   cmSepaGripperAxisZ.commandConfiguration.haltSuperimposed.jerk := -1.0;
   cmSepaGripperAxisZ.commandConfiguration.haltSuperimposed.abortAcceleration := FALSE;
   cmSepaGripperAxisZ.commandConfiguration.gearInRelative.ratioNumerator := 1;
   cmSepaGripperAxisZ.commandConfiguration.gearInRelative.ratioDenominator := 1;
   cmSepaGripperAxisZ.commandConfiguration.gearInRelative.acceleration := -1.0;
   cmSepaGripperAxisZ.commandConfiguration.gearInRelative.deceleration := -1.0;
   cmSepaGripperAxisZ.commandConfiguration.gearInRelative.jerk := -1.0;
   cmSepaGripperAxisZ.commandConfiguration.gearInRelative.ratioChangeOnTheFly := FALSE;
   cmSepaGripperAxisZ.commandConfiguration.gearInAbsolute.ratioNumerator := 1;
   cmSepaGripperAxisZ.commandConfiguration.gearInAbsolute.ratioDenominator := 1;
   cmSepaGripperAxisZ.commandConfiguration.gearInAbsolute.masterSyncPosition := 0.0;
   cmSepaGripperAxisZ.commandConfiguration.gearInAbsolute.slaveSyncPosition := 0.0;
   cmSepaGripperAxisZ.commandConfiguration.gearInAbsolute.syncProfileReference := 1;
   cmSepaGripperAxisZ.commandConfiguration.gearInAbsolute.masterStartDistance := 0.0;
   cmSepaGripperAxisZ.commandConfiguration.gearInAbsolute.velocity := -1.0;
   cmSepaGripperAxisZ.commandConfiguration.gearInAbsolute.acceleration := -1.0;
   cmSepaGripperAxisZ.commandConfiguration.gearInAbsolute.deceleration := -1.0;
   cmSepaGripperAxisZ.commandConfiguration.gearInAbsolute.jerk := -1.0;
   cmSepaGripperAxisZ.commandConfiguration.gearInAbsolute.syncDirection := 1;
   cmSepaGripperAxisZ.commandConfiguration.gearInAbsolute.ratioChangeOnTheFly := FALSE;
   cmSepaGripperAxisZ.commandConfiguration.gearInVelocity.continuousUpdate := FALSE;
   cmSepaGripperAxisZ.commandConfiguration.gearInVelocity.ratioNumerator := 1;
   cmSepaGripperAxisZ.commandConfiguration.gearInVelocity.ratioDenominator := 1;
   cmSepaGripperAxisZ.commandConfiguration.gearInVelocity.acceleration := -1.0;
   cmSepaGripperAxisZ.commandConfiguration.gearInVelocity.deceleration := -1.0;
   cmSepaGripperAxisZ.commandConfiguration.gearInVelocity.jerk := -1.0;
   cmSepaGripperAxisZ.commandConfiguration.gearInVelocity.positionControlled := FALSE;
   cmSepaGripperAxisZ.commandConfiguration.camIn.masterOffset := 0.0;
   cmSepaGripperAxisZ.commandConfiguration.camIn.slaveOffset := 0.0;
   cmSepaGripperAxisZ.commandConfiguration.camIn.masterScaling := 1.0;
   cmSepaGripperAxisZ.commandConfiguration.camIn.slaveScaling := 1.0;
   cmSepaGripperAxisZ.commandConfiguration.camIn.masterSyncPosition := 0.0;
   cmSepaGripperAxisZ.commandConfiguration.camIn.syncProfileReference := 1;
   cmSepaGripperAxisZ.commandConfiguration.camIn.masterStartDistance := 0.0;
   cmSepaGripperAxisZ.commandConfiguration.camIn.velocity := -1.0;
   cmSepaGripperAxisZ.commandConfiguration.camIn.acceleration := -1.0;
   cmSepaGripperAxisZ.commandConfiguration.camIn.deceleration := -1.0;
   cmSepaGripperAxisZ.commandConfiguration.camIn.jerk := -1.0;
   cmSepaGripperAxisZ.commandConfiguration.camIn.applicationMode := 0;
   cmSepaGripperAxisZ.commandConfiguration.camIn.syncDirection := 1;
   cmSepaGripperAxisZ.commandConfiguration.gearOutCamOut.slavePosition := 0.0;
   cmSepaGripperAxisZ.commandConfiguration.gearOutCamOut.syncProfileReference := 1;
   cmSepaGripperAxisZ.commandConfiguration.gearOutCamOut.masterStopDistance := 0.0;
   cmSepaGripperAxisZ.commandConfiguration.gearOutCamOut.deceleration := -1.0;
   cmSepaGripperAxisZ.commandConfiguration.gearOutCamOut.jerk := -1.0;
   cmSepaGripperAxisZ.commandConfiguration.gearOutCamOut.syncOutDirection := 3;
   cmSepaGripperAxisZ.commandConfiguration.gearOutCamOut.gearOutCamOutMode := -1;
   cmSepaGripperAxisZ.commandConfiguration.phasing.phaseShift := 0.0;
   cmSepaGripperAxisZ.commandConfiguration.phasing.velocity := -1.0;
   cmSepaGripperAxisZ.commandConfiguration.phasing.acceleration := -1.0;
   cmSepaGripperAxisZ.commandConfiguration.phasing.deceleration := -1.0;
   cmSepaGripperAxisZ.commandConfiguration.phasing.jerk := -1.0;
   cmSepaGripperAxisZ.commandConfiguration.phasing.profileReference := 0;
   cmSepaGripperAxisZ.commandConfiguration.phasing.phasingDistance := 0.0;
   cmSepaGripperAxisZ.commandConfiguration.phasing.startPosition := 0.0;
   cmSepaGripperAxisZ.commandConfiguration.phasing.direction := 3;
   cmSepaGripperAxisZ.commandConfiguration.phasing.phaseAbsolute := TRUE;
   cmSepaGripperAxisZ.commandConfiguration.phasing.phaseShiftChangeOnTheFly := FALSE;
   cmSepaGripperAxisZ.commandConfiguration.offset.offset := 0.0;
   cmSepaGripperAxisZ.commandConfiguration.offset.profileReference := 1;
   cmSepaGripperAxisZ.commandConfiguration.offset.offsetDistance := 0.0;
   cmSepaGripperAxisZ.commandConfiguration.offset.startPosition := 0.0;
   cmSepaGripperAxisZ.commandConfiguration.offset.direction := 3;
   cmSepaGripperAxisZ.commandConfiguration.offset.offsetAbsolute := TRUE;
   cmSepaGripperAxisZ.commandConfiguration.offset.offsetChangeOnTheFly := FALSE;
   cmSepaGripperAxisZ.commands.enableMasterControl := TRUE;
   cmSepaGripperAxisZ.commands.enableAxis := FALSE;
   cmSepaGripperAxisZ.commands.resetAxis := FALSE;
   cmSepaGripperAxisZ.commands.openBrake := FALSE;
   cmSepaGripperAxisZ.commands.jogForward := FALSE;
   cmSepaGripperAxisZ.commands.jogBackward := FALSE;
   cmSepaGripperAxisZ.commands.moveVelocity := FALSE;
   cmSepaGripperAxisZ.commands.stop := FALSE;
   cmSepaGripperAxisZ.commands.fastStop := FALSE;
   cmSepaGripperAxisZ.commands.torqueLimiting := FALSE;
   cmSepaGripperAxisZ.commands.homing := FALSE;
   cmSepaGripperAxisZ.commands.posRelative := FALSE;
   cmSepaGripperAxisZ.commands.posAbsolute := FALSE;
   cmSepaGripperAxisZ.commands.posSuperimposed := FALSE;
   cmSepaGripperAxisZ.commands.haltSuperimposed := FALSE;
   cmSepaGripperAxisZ.commands.selectSetPosition := -1;
   cmSepaGripperAxisZ.commands.uploadParameters := FALSE;
   cmSepaGripperAxisZ.commands.refreshConfiguration := FALSE;
   cmSepaGripperAxisZ.commands.editConfiguration := FALSE;
   cmSepaGripperAxisZ.commands.saveConfiguration := FALSE;
   cmSepaGripperAxisZ.commands.uploadCurrentTorque := FALSE;
   cmSepaGripperAxisZ.commands.reset := FALSE;
   cmSepaGripperAxisZ.monitoring.enable := TRUE;
   cmSepaGripperAxisZ.monitoring.referenceDesignator := WSTRING#'SepaGripperAxisZ';
   cmSepaGripperAxisZ.monitoring.enabled := TRUE;
   cmSepaGripperAxisZ.monitoring.enableManualCmds := FALSE;
   cmSepaGripperAxisZ.monitoring.reset := FALSE;
   cmSepaGripperAxisZ.monitoring.resetAxis := FALSE;
   cmSepaGripperAxisZ.monitoring.enableAxis := TRUE;
   cmSepaGripperAxisZ.monitoring.openBrake := FALSE;
   cmSepaGripperAxisZ.monitoring.jogBackward := FALSE;
   cmSepaGripperAxisZ.monitoring.jogForward := FALSE;
   cmSepaGripperAxisZ.monitoring.moveVelocity := FALSE;
   cmSepaGripperAxisZ.monitoring.stop := FALSE;
   cmSepaGripperAxisZ.monitoring.fastStop := FALSE;
   cmSepaGripperAxisZ.monitoring.torqueLimiting := FALSE;
   cmSepaGripperAxisZ.monitoring.homing := FALSE;
   cmSepaGripperAxisZ.monitoring.posRelative := FALSE;
   cmSepaGripperAxisZ.monitoring.posAbsolute := FALSE;
   cmSepaGripperAxisZ.monitoring.posSuperimposed := FALSE;
   cmSepaGripperAxisZ.monitoring.haltSuperimposed := FALSE;
   cmSepaGripperAxisZ.monitoring.brakeOpened := FALSE;
   cmSepaGripperAxisZ.monitoring.axisEnabled := TRUE;
   cmSepaGripperAxisZ.monitoring.resetActive := FALSE;
   cmSepaGripperAxisZ.monitoring.inVelocity := FALSE;
   cmSepaGripperAxisZ.monitoring.inLimitation := FALSE;
   cmSepaGripperAxisZ.monitoring.inClamping := FALSE;
   cmSepaGripperAxisZ.monitoring.startSync := FALSE;
   cmSepaGripperAxisZ.monitoring.inSync := FALSE;
   cmSepaGripperAxisZ.monitoring.inSimulation := FALSE;
   cmSepaGripperAxisZ.monitoring.jogSelected := FALSE;
   cmSepaGripperAxisZ.monitoring.moveVelocitySelected := FALSE;
   cmSepaGripperAxisZ.monitoring.stopSelected := FALSE;
   cmSepaGripperAxisZ.monitoring.fastStopSelected := FALSE;
   cmSepaGripperAxisZ.monitoring.torqueLimitingSelected := FALSE;
   cmSepaGripperAxisZ.monitoring.homingSelected := FALSE;
   cmSepaGripperAxisZ.monitoring.posRelativeSelected := FALSE;
   cmSepaGripperAxisZ.monitoring.posAbsoluteSelected := FALSE;
   cmSepaGripperAxisZ.monitoring.posSuperimposedSelected := FALSE;
   cmSepaGripperAxisZ.monitoring.haltSuperimposedSelected := FALSE;
   cmSepaGripperAxisZ.monitoring.commandBusy := FALSE;
   cmSepaGripperAxisZ.monitoring.commandDone := FALSE;
   cmSepaGripperAxisZ.monitoring.commandAborted := FALSE;
   cmSepaGripperAxisZ.monitoring.homingCommandBusy := FALSE;
   cmSepaGripperAxisZ.monitoring.homingCommandDone := FALSE;
   cmSepaGripperAxisZ.monitoring.homingCommandAborted := FALSE;
   cmSepaGripperAxisZ.monitoring.superimposedBusy := FALSE;
   cmSepaGripperAxisZ.monitoring.superimposedDone := FALSE;
   cmSepaGripperAxisZ.monitoring.superimposedAborted := FALSE;
   cmSepaGripperAxisZ.monitoring.selectSetPosition := -1;
   cmSepaGripperAxisZ.monitoring.selectionController := FALSE;
   cmSepaGripperAxisZ.monitoring.interlockGeneral := TRUE;
   cmSepaGripperAxisZ.monitoring.interlockJogForward := TRUE;
   cmSepaGripperAxisZ.monitoring.interlockJogBackward := TRUE;
   cmSepaGripperAxisZ.monitoring.interlockWarningGeneral := FALSE;
   cmSepaGripperAxisZ.monitoring.interlockWarningJogForward := FALSE;
   cmSepaGripperAxisZ.monitoring.interlockWarningJogBackward := FALSE;
   cmSepaGripperAxisZ.monitoring.valid := TRUE;
   cmSepaGripperAxisZ.monitoring.busy := TRUE;
   cmSepaGripperAxisZ.monitoring.error := FALSE;
   cmSepaGripperAxisZ.monitoring.status := 16#7002;
   cmSepaGripperAxisZ.monitoring.subfunctionStatus := 16#0000;
   cmSepaGripperAxisZ.monitoring.actualPosition := 0.0;
   cmSepaGripperAxisZ.monitoring.actualSpeed := 0.0;
   cmSepaGripperAxisZ.monitoring.speedUnit := 1062;
   cmSepaGripperAxisZ.monitoring.positionUnit := 1013;
   cmSepaGripperAxisZ.monitoring.axisStatus1 := 16#0200_10E1;
   cmSepaGripperAxisZ.monitoring.axisStatus2 := 16#0000_0000;
   cmSepaGripperAxisZ.monitoring.axisType := 1;
   cmSepaGripperAxisZ.monitoring.maxVelocity := 2500.0;
   cmSepaGripperAxisZ.monitoring.actualCurrent := 0.0;
   cmSepaGripperAxisZ.monitoring.actualTorque := 0.0;
   cmSepaGripperAxisZ.monitoring.velocityOverrideEnabled := FALSE;
   cmSepaGripperAxisZ.monitoring.sinaParaError := FALSE;
   cmSepaGripperAxisZ.monitoring.sinaParaStatus := 16#0000_0000;
   cmSepaGripperAxisZ.configuration.referenceDesignator := WSTRING#'SepaGripperAxisZ';
   cmSepaGripperAxisZ.configuration.disableAlarms := FALSE;
   cmSepaGripperAxisZ.configuration.masterControlPopUp := TRUE;
   cmSepaGripperAxisZ.configuration.setPositions[0].position := 0.0;
   cmSepaGripperAxisZ.configuration.setPositions[1].position := 25.0;
   cmSepaGripperAxisZ.configuration.setPositions[2].position := 2.0;
   cmSepaGripperAxisZ.configuration.setPositions[3].position := 3.0;
   cmSepaGripperAxisZ.configuration.setPositions[4].position := 4.0;
   cmSepaGripperAxisZ.configuration.setPositions[5].position := 5.0;
   cmSepaGripperAxisZ.configuration.setPositions[6].position := 50.0;
   cmSepaGripperAxisZ.configuration.setPositions[7..15].position := 0.0;
   cmSepaGripperAxisZ.configuration.setPositions[0..6].velocity := 50.0;
   cmSepaGripperAxisZ.configuration.setPositions[7..15].velocity := -1.0;
   cmSepaGripperAxisZ.configuration.setPositions[0..6].acceleration := 500.0;
   cmSepaGripperAxisZ.configuration.setPositions[7..15].acceleration := -1.0;
   cmSepaGripperAxisZ.configuration.setPositions[0..6].deceleration := 500.0;
   cmSepaGripperAxisZ.configuration.setPositions[7..15].deceleration := -1.0;
   cmSepaGripperAxisZ.configuration.setPositions[0..15]."name" := '';
   cmSepaGripperAxisC.commandConfiguration.generalSettings.stopOnError := TRUE;
   cmSepaGripperAxisC.commandConfiguration.generalSettings.resetWithRestart := FALSE;
   cmSepaGripperAxisC.commandConfiguration.generalSettings.abortWaitingSyncCmd := TRUE;
   cmSepaGripperAxisC.commandConfiguration.power.startMode := 1;
   cmSepaGripperAxisC.commandConfiguration.power.stopMode := 0;
   cmSepaGripperAxisC.commandConfiguration.power.syncMotionSimulation := FALSE;
   cmSepaGripperAxisC.commandConfiguration.power.syncMotionSimulationExtendedMode := -1;
   cmSepaGripperAxisC.commandConfiguration.jog.velocity := 0.0;
   cmSepaGripperAxisC.commandConfiguration.jog.acceleration := -1.0;
   cmSepaGripperAxisC.commandConfiguration.jog.deceleration := -1.0;
   cmSepaGripperAxisC.commandConfiguration.jog.jerk := -1.0;
   cmSepaGripperAxisC.commandConfiguration.jog.positionControlled := TRUE;
   cmSepaGripperAxisC.commandConfiguration.jog.increment := 0.0;
   cmSepaGripperAxisC.commandConfiguration.jog.mode := 0;
   cmSepaGripperAxisC.commandConfiguration.moveVelocity.velocity := 0.0;
   cmSepaGripperAxisC.commandConfiguration.moveVelocity.acceleration := -1.0;
   cmSepaGripperAxisC.commandConfiguration.moveVelocity.deceleration := -1.0;
   cmSepaGripperAxisC.commandConfiguration.moveVelocity.jerk := -1.0;
   cmSepaGripperAxisC.commandConfiguration.moveVelocity.direction := 0;
   cmSepaGripperAxisC.commandConfiguration.moveVelocity.positionControlled := TRUE;
   cmSepaGripperAxisC.commandConfiguration.moveVelocity.velocityChangeOnTheFly := FALSE;
   cmSepaGripperAxisC.commandConfiguration.stop.deceleration := -1.0;
   cmSepaGripperAxisC.commandConfiguration.stop.jerk := -1.0;
   cmSepaGripperAxisC.commandConfiguration.stop.abortAcceleration := FALSE;
   cmSepaGripperAxisC.commandConfiguration.fastStop.deceleration := -1.0;
   cmSepaGripperAxisC.commandConfiguration.fastStop.jerk := -1.0;
   cmSepaGripperAxisC.commandConfiguration.fastStop.abortAcceleration := FALSE;
   cmSepaGripperAxisC.commandConfiguration.fastStop.replaceStopPossible := FALSE;
   cmSepaGripperAxisC.commandConfiguration.torqueLimiting.limit := -1.0;
   cmSepaGripperAxisC.commandConfiguration.torqueLimiting.mode := 0;
   cmSepaGripperAxisC.commandConfiguration.homing.position := 0.0;
   cmSepaGripperAxisC.commandConfiguration.homing.mode := 0;
   cmSepaGripperAxisC.commandConfiguration.homing.sensor := 0;
   cmSepaGripperAxisC.commandConfiguration.homing.extendedMode := -1;
   cmSepaGripperAxisC.commandConfiguration.homing.extendedModeTorqueLimit := 0.0;
   cmSepaGripperAxisC.commandConfiguration.homing.extendedModeTargetPosition := 0.0;
   cmSepaGripperAxisC.commandConfiguration.posRelative.distance := 0.0;
   cmSepaGripperAxisC.commandConfiguration.posRelative.velocity := -1.0;
   cmSepaGripperAxisC.commandConfiguration.posRelative.acceleration := -1.0;
   cmSepaGripperAxisC.commandConfiguration.posRelative.deceleration := -1.0;
   cmSepaGripperAxisC.commandConfiguration.posRelative.jerk := -1.0;
   cmSepaGripperAxisC.commandConfiguration.posRelative.direction := 0;
   cmSepaGripperAxisC.commandConfiguration.posAbsolute.position := 0.0;
   cmSepaGripperAxisC.commandConfiguration.posAbsolute.velocity := -1.0;
   cmSepaGripperAxisC.commandConfiguration.posAbsolute.acceleration := -1.0;
   cmSepaGripperAxisC.commandConfiguration.posAbsolute.deceleration := -1.0;
   cmSepaGripperAxisC.commandConfiguration.posAbsolute.jerk := -1.0;
   cmSepaGripperAxisC.commandConfiguration.posAbsolute.direction := 1;
   cmSepaGripperAxisC.commandConfiguration.posAbsolute.positionChangeOnTheFly := FALSE;
   cmSepaGripperAxisC.commandConfiguration.posAbsolute.velocityChangeOnTheFly := FALSE;
   cmSepaGripperAxisC.commandConfiguration.posSuperimposed.distance := 0.0;
   cmSepaGripperAxisC.commandConfiguration.posSuperimposed.velocityDiff := -1.0;
   cmSepaGripperAxisC.commandConfiguration.posSuperimposed.acceleration := -1.0;
   cmSepaGripperAxisC.commandConfiguration.posSuperimposed.deceleration := -1.0;
   cmSepaGripperAxisC.commandConfiguration.posSuperimposed.jerk := -1.0;
   cmSepaGripperAxisC.commandConfiguration.posSuperimposed.direction := 0;
   cmSepaGripperAxisC.commandConfiguration.haltSuperimposed.deceleration := -1.0;
   cmSepaGripperAxisC.commandConfiguration.haltSuperimposed.jerk := -1.0;
   cmSepaGripperAxisC.commandConfiguration.haltSuperimposed.abortAcceleration := FALSE;
   cmSepaGripperAxisC.commandConfiguration.gearInRelative.ratioNumerator := 1;
   cmSepaGripperAxisC.commandConfiguration.gearInRelative.ratioDenominator := 1;
   cmSepaGripperAxisC.commandConfiguration.gearInRelative.acceleration := -1.0;
   cmSepaGripperAxisC.commandConfiguration.gearInRelative.deceleration := -1.0;
   cmSepaGripperAxisC.commandConfiguration.gearInRelative.jerk := -1.0;
   cmSepaGripperAxisC.commandConfiguration.gearInRelative.ratioChangeOnTheFly := FALSE;
   cmSepaGripperAxisC.commandConfiguration.gearInAbsolute.ratioNumerator := 1;
   cmSepaGripperAxisC.commandConfiguration.gearInAbsolute.ratioDenominator := 1;
   cmSepaGripperAxisC.commandConfiguration.gearInAbsolute.masterSyncPosition := 0.0;
   cmSepaGripperAxisC.commandConfiguration.gearInAbsolute.slaveSyncPosition := 0.0;
   cmSepaGripperAxisC.commandConfiguration.gearInAbsolute.syncProfileReference := 1;
   cmSepaGripperAxisC.commandConfiguration.gearInAbsolute.masterStartDistance := 0.0;
   cmSepaGripperAxisC.commandConfiguration.gearInAbsolute.velocity := -1.0;
   cmSepaGripperAxisC.commandConfiguration.gearInAbsolute.acceleration := -1.0;
   cmSepaGripperAxisC.commandConfiguration.gearInAbsolute.deceleration := -1.0;
   cmSepaGripperAxisC.commandConfiguration.gearInAbsolute.jerk := -1.0;
   cmSepaGripperAxisC.commandConfiguration.gearInAbsolute.syncDirection := 1;
   cmSepaGripperAxisC.commandConfiguration.gearInAbsolute.ratioChangeOnTheFly := FALSE;
   cmSepaGripperAxisC.commandConfiguration.gearInVelocity.continuousUpdate := FALSE;
   cmSepaGripperAxisC.commandConfiguration.gearInVelocity.ratioNumerator := 1;
   cmSepaGripperAxisC.commandConfiguration.gearInVelocity.ratioDenominator := 1;
   cmSepaGripperAxisC.commandConfiguration.gearInVelocity.acceleration := -1.0;
   cmSepaGripperAxisC.commandConfiguration.gearInVelocity.deceleration := -1.0;
   cmSepaGripperAxisC.commandConfiguration.gearInVelocity.jerk := -1.0;
   cmSepaGripperAxisC.commandConfiguration.gearInVelocity.positionControlled := FALSE;
   cmSepaGripperAxisC.commandConfiguration.camIn.masterOffset := 0.0;
   cmSepaGripperAxisC.commandConfiguration.camIn.slaveOffset := 0.0;
   cmSepaGripperAxisC.commandConfiguration.camIn.masterScaling := 1.0;
   cmSepaGripperAxisC.commandConfiguration.camIn.slaveScaling := 1.0;
   cmSepaGripperAxisC.commandConfiguration.camIn.masterSyncPosition := 0.0;
   cmSepaGripperAxisC.commandConfiguration.camIn.syncProfileReference := 1;
   cmSepaGripperAxisC.commandConfiguration.camIn.masterStartDistance := 0.0;
   cmSepaGripperAxisC.commandConfiguration.camIn.velocity := -1.0;
   cmSepaGripperAxisC.commandConfiguration.camIn.acceleration := -1.0;
   cmSepaGripperAxisC.commandConfiguration.camIn.deceleration := -1.0;
   cmSepaGripperAxisC.commandConfiguration.camIn.jerk := -1.0;
   cmSepaGripperAxisC.commandConfiguration.camIn.applicationMode := 0;
   cmSepaGripperAxisC.commandConfiguration.camIn.syncDirection := 1;
   cmSepaGripperAxisC.commandConfiguration.gearOutCamOut.slavePosition := 0.0;
   cmSepaGripperAxisC.commandConfiguration.gearOutCamOut.syncProfileReference := 1;
   cmSepaGripperAxisC.commandConfiguration.gearOutCamOut.masterStopDistance := 0.0;
   cmSepaGripperAxisC.commandConfiguration.gearOutCamOut.deceleration := -1.0;
   cmSepaGripperAxisC.commandConfiguration.gearOutCamOut.jerk := -1.0;
   cmSepaGripperAxisC.commandConfiguration.gearOutCamOut.syncOutDirection := 3;
   cmSepaGripperAxisC.commandConfiguration.gearOutCamOut.gearOutCamOutMode := -1;
   cmSepaGripperAxisC.commandConfiguration.phasing.phaseShift := 0.0;
   cmSepaGripperAxisC.commandConfiguration.phasing.velocity := -1.0;
   cmSepaGripperAxisC.commandConfiguration.phasing.acceleration := -1.0;
   cmSepaGripperAxisC.commandConfiguration.phasing.deceleration := -1.0;
   cmSepaGripperAxisC.commandConfiguration.phasing.jerk := -1.0;
   cmSepaGripperAxisC.commandConfiguration.phasing.profileReference := 0;
   cmSepaGripperAxisC.commandConfiguration.phasing.phasingDistance := 0.0;
   cmSepaGripperAxisC.commandConfiguration.phasing.startPosition := 0.0;
   cmSepaGripperAxisC.commandConfiguration.phasing.direction := 3;
   cmSepaGripperAxisC.commandConfiguration.phasing.phaseAbsolute := TRUE;
   cmSepaGripperAxisC.commandConfiguration.phasing.phaseShiftChangeOnTheFly := FALSE;
   cmSepaGripperAxisC.commandConfiguration.offset.offset := 0.0;
   cmSepaGripperAxisC.commandConfiguration.offset.profileReference := 1;
   cmSepaGripperAxisC.commandConfiguration.offset.offsetDistance := 0.0;
   cmSepaGripperAxisC.commandConfiguration.offset.startPosition := 0.0;
   cmSepaGripperAxisC.commandConfiguration.offset.direction := 3;
   cmSepaGripperAxisC.commandConfiguration.offset.offsetAbsolute := TRUE;
   cmSepaGripperAxisC.commandConfiguration.offset.offsetChangeOnTheFly := FALSE;
   cmSepaGripperAxisC.commands.enableMasterControl := TRUE;
   cmSepaGripperAxisC.commands.enableAxis := FALSE;
   cmSepaGripperAxisC.commands.resetAxis := FALSE;
   cmSepaGripperAxisC.commands.openBrake := FALSE;
   cmSepaGripperAxisC.commands.jogForward := FALSE;
   cmSepaGripperAxisC.commands.jogBackward := FALSE;
   cmSepaGripperAxisC.commands.moveVelocity := FALSE;
   cmSepaGripperAxisC.commands.stop := FALSE;
   cmSepaGripperAxisC.commands.fastStop := FALSE;
   cmSepaGripperAxisC.commands.torqueLimiting := FALSE;
   cmSepaGripperAxisC.commands.homing := FALSE;
   cmSepaGripperAxisC.commands.posRelative := FALSE;
   cmSepaGripperAxisC.commands.posAbsolute := FALSE;
   cmSepaGripperAxisC.commands.posSuperimposed := FALSE;
   cmSepaGripperAxisC.commands.haltSuperimposed := FALSE;
   cmSepaGripperAxisC.commands.selectSetPosition := -1;
   cmSepaGripperAxisC.commands.uploadParameters := FALSE;
   cmSepaGripperAxisC.commands.refreshConfiguration := FALSE;
   cmSepaGripperAxisC.commands.editConfiguration := FALSE;
   cmSepaGripperAxisC.commands.saveConfiguration := FALSE;
   cmSepaGripperAxisC.commands.uploadCurrentTorque := FALSE;
   cmSepaGripperAxisC.commands.reset := FALSE;
   cmSepaGripperAxisC.monitoring.enable := TRUE;
   cmSepaGripperAxisC.monitoring.referenceDesignator := WSTRING#'SepaGripperAxisC';
   cmSepaGripperAxisC.monitoring.enabled := TRUE;
   cmSepaGripperAxisC.monitoring.enableManualCmds := FALSE;
   cmSepaGripperAxisC.monitoring.reset := FALSE;
   cmSepaGripperAxisC.monitoring.resetAxis := FALSE;
   cmSepaGripperAxisC.monitoring.enableAxis := TRUE;
   cmSepaGripperAxisC.monitoring.openBrake := FALSE;
   cmSepaGripperAxisC.monitoring.jogBackward := FALSE;
   cmSepaGripperAxisC.monitoring.jogForward := FALSE;
   cmSepaGripperAxisC.monitoring.moveVelocity := FALSE;
   cmSepaGripperAxisC.monitoring.stop := FALSE;
   cmSepaGripperAxisC.monitoring.fastStop := FALSE;
   cmSepaGripperAxisC.monitoring.torqueLimiting := FALSE;
   cmSepaGripperAxisC.monitoring.homing := FALSE;
   cmSepaGripperAxisC.monitoring.posRelative := FALSE;
   cmSepaGripperAxisC.monitoring.posAbsolute := FALSE;
   cmSepaGripperAxisC.monitoring.posSuperimposed := FALSE;
   cmSepaGripperAxisC.monitoring.haltSuperimposed := FALSE;
   cmSepaGripperAxisC.monitoring.brakeOpened := FALSE;
   cmSepaGripperAxisC.monitoring.axisEnabled := TRUE;
   cmSepaGripperAxisC.monitoring.resetActive := FALSE;
   cmSepaGripperAxisC.monitoring.inVelocity := FALSE;
   cmSepaGripperAxisC.monitoring.inLimitation := FALSE;
   cmSepaGripperAxisC.monitoring.inClamping := FALSE;
   cmSepaGripperAxisC.monitoring.startSync := FALSE;
   cmSepaGripperAxisC.monitoring.inSync := FALSE;
   cmSepaGripperAxisC.monitoring.inSimulation := FALSE;
   cmSepaGripperAxisC.monitoring.jogSelected := FALSE;
   cmSepaGripperAxisC.monitoring.moveVelocitySelected := FALSE;
   cmSepaGripperAxisC.monitoring.stopSelected := FALSE;
   cmSepaGripperAxisC.monitoring.fastStopSelected := FALSE;
   cmSepaGripperAxisC.monitoring.torqueLimitingSelected := FALSE;
   cmSepaGripperAxisC.monitoring.homingSelected := FALSE;
   cmSepaGripperAxisC.monitoring.posRelativeSelected := FALSE;
   cmSepaGripperAxisC.monitoring.posAbsoluteSelected := FALSE;
   cmSepaGripperAxisC.monitoring.posSuperimposedSelected := FALSE;
   cmSepaGripperAxisC.monitoring.haltSuperimposedSelected := FALSE;
   cmSepaGripperAxisC.monitoring.commandBusy := FALSE;
   cmSepaGripperAxisC.monitoring.commandDone := FALSE;
   cmSepaGripperAxisC.monitoring.commandAborted := FALSE;
   cmSepaGripperAxisC.monitoring.homingCommandBusy := FALSE;
   cmSepaGripperAxisC.monitoring.homingCommandDone := FALSE;
   cmSepaGripperAxisC.monitoring.homingCommandAborted := FALSE;
   cmSepaGripperAxisC.monitoring.superimposedBusy := FALSE;
   cmSepaGripperAxisC.monitoring.superimposedDone := FALSE;
   cmSepaGripperAxisC.monitoring.superimposedAborted := FALSE;
   cmSepaGripperAxisC.monitoring.selectSetPosition := -1;
   cmSepaGripperAxisC.monitoring.selectionController := FALSE;
   cmSepaGripperAxisC.monitoring.interlockGeneral := TRUE;
   cmSepaGripperAxisC.monitoring.interlockJogForward := TRUE;
   cmSepaGripperAxisC.monitoring.interlockJogBackward := TRUE;
   cmSepaGripperAxisC.monitoring.interlockWarningGeneral := FALSE;
   cmSepaGripperAxisC.monitoring.interlockWarningJogForward := FALSE;
   cmSepaGripperAxisC.monitoring.interlockWarningJogBackward := FALSE;
   cmSepaGripperAxisC.monitoring.valid := TRUE;
   cmSepaGripperAxisC.monitoring.busy := TRUE;
   cmSepaGripperAxisC.monitoring.error := FALSE;
   cmSepaGripperAxisC.monitoring.status := 16#7002;
   cmSepaGripperAxisC.monitoring.subfunctionStatus := 16#0000;
   cmSepaGripperAxisC.monitoring.actualPosition := 0.0;
   cmSepaGripperAxisC.monitoring.actualSpeed := 0.0;
   cmSepaGripperAxisC.monitoring.speedUnit := 1521;
   cmSepaGripperAxisC.monitoring.positionUnit := 1005;
   cmSepaGripperAxisC.monitoring.axisStatus1 := 16#0200_10E1;
   cmSepaGripperAxisC.monitoring.axisStatus2 := 16#0000_0000;
   cmSepaGripperAxisC.monitoring.axisType := 1;
   cmSepaGripperAxisC.monitoring.maxVelocity := 18000.0;
   cmSepaGripperAxisC.monitoring.actualCurrent := 0.0;
   cmSepaGripperAxisC.monitoring.actualTorque := 0.0;
   cmSepaGripperAxisC.monitoring.velocityOverrideEnabled := FALSE;
   cmSepaGripperAxisC.monitoring.sinaParaError := FALSE;
   cmSepaGripperAxisC.monitoring.sinaParaStatus := 16#0000_0000;
   cmSepaGripperAxisC.configuration.referenceDesignator := WSTRING#'SepaGripperAxisC';
   cmSepaGripperAxisC.configuration.disableAlarms := FALSE;
   cmSepaGripperAxisC.configuration.masterControlPopUp := TRUE;
   cmSepaGripperAxisC.configuration.setPositions[0].position := 0.0;
   cmSepaGripperAxisC.configuration.setPositions[1].position := 180.0;
   cmSepaGripperAxisC.configuration.setPositions[2].position := 90.0;
   cmSepaGripperAxisC.configuration.setPositions[3..15].position := 0.0;
   cmSepaGripperAxisC.configuration.setPositions[0..2].velocity := 100.0;
   cmSepaGripperAxisC.configuration.setPositions[3..15].velocity := -1.0;
   cmSepaGripperAxisC.configuration.setPositions[0..2].acceleration := 1000.0;
   cmSepaGripperAxisC.configuration.setPositions[3..15].acceleration := -1.0;
   cmSepaGripperAxisC.configuration.setPositions[0..2].deceleration := 1000.0;
   cmSepaGripperAxisC.configuration.setPositions[3..15].deceleration := -1.0;
   cmSepaGripperAxisC.configuration.setPositions[0..15]."name" := '';
   cmJRWinderRearAxisY.commandConfiguration.generalSettings.stopOnError := TRUE;
   cmJRWinderRearAxisY.commandConfiguration.generalSettings.resetWithRestart := FALSE;
   cmJRWinderRearAxisY.commandConfiguration.generalSettings.abortWaitingSyncCmd := TRUE;
   cmJRWinderRearAxisY.commandConfiguration.power.startMode := 1;
   cmJRWinderRearAxisY.commandConfiguration.power.stopMode := 0;
   cmJRWinderRearAxisY.commandConfiguration.power.syncMotionSimulation := FALSE;
   cmJRWinderRearAxisY.commandConfiguration.power.syncMotionSimulationExtendedMode := -1;
   cmJRWinderRearAxisY.commandConfiguration.jog.velocity := 0.0;
   cmJRWinderRearAxisY.commandConfiguration.jog.acceleration := -1.0;
   cmJRWinderRearAxisY.commandConfiguration.jog.deceleration := -1.0;
   cmJRWinderRearAxisY.commandConfiguration.jog.jerk := -1.0;
   cmJRWinderRearAxisY.commandConfiguration.jog.positionControlled := TRUE;
   cmJRWinderRearAxisY.commandConfiguration.jog.increment := 0.0;
   cmJRWinderRearAxisY.commandConfiguration.jog.mode := 0;
   cmJRWinderRearAxisY.commandConfiguration.moveVelocity.velocity := 0.0;
   cmJRWinderRearAxisY.commandConfiguration.moveVelocity.acceleration := -1.0;
   cmJRWinderRearAxisY.commandConfiguration.moveVelocity.deceleration := -1.0;
   cmJRWinderRearAxisY.commandConfiguration.moveVelocity.jerk := -1.0;
   cmJRWinderRearAxisY.commandConfiguration.moveVelocity.direction := 0;
   cmJRWinderRearAxisY.commandConfiguration.moveVelocity.positionControlled := TRUE;
   cmJRWinderRearAxisY.commandConfiguration.moveVelocity.velocityChangeOnTheFly := FALSE;
   cmJRWinderRearAxisY.commandConfiguration.stop.deceleration := -1.0;
   cmJRWinderRearAxisY.commandConfiguration.stop.jerk := -1.0;
   cmJRWinderRearAxisY.commandConfiguration.stop.abortAcceleration := FALSE;
   cmJRWinderRearAxisY.commandConfiguration.fastStop.deceleration := -1.0;
   cmJRWinderRearAxisY.commandConfiguration.fastStop.jerk := -1.0;
   cmJRWinderRearAxisY.commandConfiguration.fastStop.abortAcceleration := FALSE;
   cmJRWinderRearAxisY.commandConfiguration.fastStop.replaceStopPossible := FALSE;
   cmJRWinderRearAxisY.commandConfiguration.torqueLimiting.limit := -1.0;
   cmJRWinderRearAxisY.commandConfiguration.torqueLimiting.mode := 0;
   cmJRWinderRearAxisY.commandConfiguration.homing.position := 0.0;
   cmJRWinderRearAxisY.commandConfiguration.homing.mode := 0;
   cmJRWinderRearAxisY.commandConfiguration.homing.sensor := 0;
   cmJRWinderRearAxisY.commandConfiguration.homing.extendedMode := -1;
   cmJRWinderRearAxisY.commandConfiguration.homing.extendedModeTorqueLimit := 0.0;
   cmJRWinderRearAxisY.commandConfiguration.homing.extendedModeTargetPosition := 0.0;
   cmJRWinderRearAxisY.commandConfiguration.posRelative.distance := 0.0;
   cmJRWinderRearAxisY.commandConfiguration.posRelative.velocity := -1.0;
   cmJRWinderRearAxisY.commandConfiguration.posRelative.acceleration := -1.0;
   cmJRWinderRearAxisY.commandConfiguration.posRelative.deceleration := -1.0;
   cmJRWinderRearAxisY.commandConfiguration.posRelative.jerk := -1.0;
   cmJRWinderRearAxisY.commandConfiguration.posRelative.direction := 0;
   cmJRWinderRearAxisY.commandConfiguration.posAbsolute.position := 0.0;
   cmJRWinderRearAxisY.commandConfiguration.posAbsolute.velocity := -1.0;
   cmJRWinderRearAxisY.commandConfiguration.posAbsolute.acceleration := -1.0;
   cmJRWinderRearAxisY.commandConfiguration.posAbsolute.deceleration := -1.0;
   cmJRWinderRearAxisY.commandConfiguration.posAbsolute.jerk := -1.0;
   cmJRWinderRearAxisY.commandConfiguration.posAbsolute.direction := 1;
   cmJRWinderRearAxisY.commandConfiguration.posAbsolute.positionChangeOnTheFly := FALSE;
   cmJRWinderRearAxisY.commandConfiguration.posAbsolute.velocityChangeOnTheFly := FALSE;
   cmJRWinderRearAxisY.commandConfiguration.posSuperimposed.distance := 0.0;
   cmJRWinderRearAxisY.commandConfiguration.posSuperimposed.velocityDiff := -1.0;
   cmJRWinderRearAxisY.commandConfiguration.posSuperimposed.acceleration := -1.0;
   cmJRWinderRearAxisY.commandConfiguration.posSuperimposed.deceleration := -1.0;
   cmJRWinderRearAxisY.commandConfiguration.posSuperimposed.jerk := -1.0;
   cmJRWinderRearAxisY.commandConfiguration.posSuperimposed.direction := 0;
   cmJRWinderRearAxisY.commandConfiguration.haltSuperimposed.deceleration := -1.0;
   cmJRWinderRearAxisY.commandConfiguration.haltSuperimposed.jerk := -1.0;
   cmJRWinderRearAxisY.commandConfiguration.haltSuperimposed.abortAcceleration := FALSE;
   cmJRWinderRearAxisY.commandConfiguration.gearInRelative.ratioNumerator := 1;
   cmJRWinderRearAxisY.commandConfiguration.gearInRelative.ratioDenominator := 1;
   cmJRWinderRearAxisY.commandConfiguration.gearInRelative.acceleration := -1.0;
   cmJRWinderRearAxisY.commandConfiguration.gearInRelative.deceleration := -1.0;
   cmJRWinderRearAxisY.commandConfiguration.gearInRelative.jerk := -1.0;
   cmJRWinderRearAxisY.commandConfiguration.gearInRelative.ratioChangeOnTheFly := FALSE;
   cmJRWinderRearAxisY.commandConfiguration.gearInAbsolute.ratioNumerator := 1;
   cmJRWinderRearAxisY.commandConfiguration.gearInAbsolute.ratioDenominator := 1;
   cmJRWinderRearAxisY.commandConfiguration.gearInAbsolute.masterSyncPosition := 0.0;
   cmJRWinderRearAxisY.commandConfiguration.gearInAbsolute.slaveSyncPosition := 0.0;
   cmJRWinderRearAxisY.commandConfiguration.gearInAbsolute.syncProfileReference := 1;
   cmJRWinderRearAxisY.commandConfiguration.gearInAbsolute.masterStartDistance := 0.0;
   cmJRWinderRearAxisY.commandConfiguration.gearInAbsolute.velocity := -1.0;
   cmJRWinderRearAxisY.commandConfiguration.gearInAbsolute.acceleration := -1.0;
   cmJRWinderRearAxisY.commandConfiguration.gearInAbsolute.deceleration := -1.0;
   cmJRWinderRearAxisY.commandConfiguration.gearInAbsolute.jerk := -1.0;
   cmJRWinderRearAxisY.commandConfiguration.gearInAbsolute.syncDirection := 1;
   cmJRWinderRearAxisY.commandConfiguration.gearInAbsolute.ratioChangeOnTheFly := FALSE;
   cmJRWinderRearAxisY.commandConfiguration.gearInVelocity.continuousUpdate := FALSE;
   cmJRWinderRearAxisY.commandConfiguration.gearInVelocity.ratioNumerator := 1;
   cmJRWinderRearAxisY.commandConfiguration.gearInVelocity.ratioDenominator := 1;
   cmJRWinderRearAxisY.commandConfiguration.gearInVelocity.acceleration := -1.0;
   cmJRWinderRearAxisY.commandConfiguration.gearInVelocity.deceleration := -1.0;
   cmJRWinderRearAxisY.commandConfiguration.gearInVelocity.jerk := -1.0;
   cmJRWinderRearAxisY.commandConfiguration.gearInVelocity.positionControlled := FALSE;
   cmJRWinderRearAxisY.commandConfiguration.camIn.masterOffset := 0.0;
   cmJRWinderRearAxisY.commandConfiguration.camIn.slaveOffset := 0.0;
   cmJRWinderRearAxisY.commandConfiguration.camIn.masterScaling := 1.0;
   cmJRWinderRearAxisY.commandConfiguration.camIn.slaveScaling := 1.0;
   cmJRWinderRearAxisY.commandConfiguration.camIn.masterSyncPosition := 0.0;
   cmJRWinderRearAxisY.commandConfiguration.camIn.syncProfileReference := 1;
   cmJRWinderRearAxisY.commandConfiguration.camIn.masterStartDistance := 0.0;
   cmJRWinderRearAxisY.commandConfiguration.camIn.velocity := -1.0;
   cmJRWinderRearAxisY.commandConfiguration.camIn.acceleration := -1.0;
   cmJRWinderRearAxisY.commandConfiguration.camIn.deceleration := -1.0;
   cmJRWinderRearAxisY.commandConfiguration.camIn.jerk := -1.0;
   cmJRWinderRearAxisY.commandConfiguration.camIn.applicationMode := 0;
   cmJRWinderRearAxisY.commandConfiguration.camIn.syncDirection := 1;
   cmJRWinderRearAxisY.commandConfiguration.gearOutCamOut.slavePosition := 0.0;
   cmJRWinderRearAxisY.commandConfiguration.gearOutCamOut.syncProfileReference := 1;
   cmJRWinderRearAxisY.commandConfiguration.gearOutCamOut.masterStopDistance := 0.0;
   cmJRWinderRearAxisY.commandConfiguration.gearOutCamOut.deceleration := -1.0;
   cmJRWinderRearAxisY.commandConfiguration.gearOutCamOut.jerk := -1.0;
   cmJRWinderRearAxisY.commandConfiguration.gearOutCamOut.syncOutDirection := 3;
   cmJRWinderRearAxisY.commandConfiguration.gearOutCamOut.gearOutCamOutMode := -1;
   cmJRWinderRearAxisY.commandConfiguration.phasing.phaseShift := 0.0;
   cmJRWinderRearAxisY.commandConfiguration.phasing.velocity := -1.0;
   cmJRWinderRearAxisY.commandConfiguration.phasing.acceleration := -1.0;
   cmJRWinderRearAxisY.commandConfiguration.phasing.deceleration := -1.0;
   cmJRWinderRearAxisY.commandConfiguration.phasing.jerk := -1.0;
   cmJRWinderRearAxisY.commandConfiguration.phasing.profileReference := 0;
   cmJRWinderRearAxisY.commandConfiguration.phasing.phasingDistance := 0.0;
   cmJRWinderRearAxisY.commandConfiguration.phasing.startPosition := 0.0;
   cmJRWinderRearAxisY.commandConfiguration.phasing.direction := 3;
   cmJRWinderRearAxisY.commandConfiguration.phasing.phaseAbsolute := TRUE;
   cmJRWinderRearAxisY.commandConfiguration.phasing.phaseShiftChangeOnTheFly := FALSE;
   cmJRWinderRearAxisY.commandConfiguration.offset.offset := 0.0;
   cmJRWinderRearAxisY.commandConfiguration.offset.profileReference := 1;
   cmJRWinderRearAxisY.commandConfiguration.offset.offsetDistance := 0.0;
   cmJRWinderRearAxisY.commandConfiguration.offset.startPosition := 0.0;
   cmJRWinderRearAxisY.commandConfiguration.offset.direction := 3;
   cmJRWinderRearAxisY.commandConfiguration.offset.offsetAbsolute := TRUE;
   cmJRWinderRearAxisY.commandConfiguration.offset.offsetChangeOnTheFly := FALSE;
   cmJRWinderRearAxisY.commands.enableMasterControl := TRUE;
   cmJRWinderRearAxisY.commands.enableAxis := FALSE;
   cmJRWinderRearAxisY.commands.resetAxis := FALSE;
   cmJRWinderRearAxisY.commands.openBrake := FALSE;
   cmJRWinderRearAxisY.commands.jogForward := FALSE;
   cmJRWinderRearAxisY.commands.jogBackward := FALSE;
   cmJRWinderRearAxisY.commands.moveVelocity := FALSE;
   cmJRWinderRearAxisY.commands.stop := FALSE;
   cmJRWinderRearAxisY.commands.fastStop := FALSE;
   cmJRWinderRearAxisY.commands.torqueLimiting := FALSE;
   cmJRWinderRearAxisY.commands.homing := FALSE;
   cmJRWinderRearAxisY.commands.posRelative := FALSE;
   cmJRWinderRearAxisY.commands.posAbsolute := FALSE;
   cmJRWinderRearAxisY.commands.posSuperimposed := FALSE;
   cmJRWinderRearAxisY.commands.haltSuperimposed := FALSE;
   cmJRWinderRearAxisY.commands.selectSetPosition := -1;
   cmJRWinderRearAxisY.commands.uploadParameters := FALSE;
   cmJRWinderRearAxisY.commands.refreshConfiguration := FALSE;
   cmJRWinderRearAxisY.commands.editConfiguration := FALSE;
   cmJRWinderRearAxisY.commands.saveConfiguration := FALSE;
   cmJRWinderRearAxisY.commands.uploadCurrentTorque := FALSE;
   cmJRWinderRearAxisY.commands.reset := FALSE;
   cmJRWinderRearAxisY.monitoring.enable := TRUE;
   cmJRWinderRearAxisY.monitoring.referenceDesignator := WSTRING#'JRWinderRearAxisY';
   cmJRWinderRearAxisY.monitoring.enabled := TRUE;
   cmJRWinderRearAxisY.monitoring.enableManualCmds := FALSE;
   cmJRWinderRearAxisY.monitoring.reset := FALSE;
   cmJRWinderRearAxisY.monitoring.resetAxis := FALSE;
   cmJRWinderRearAxisY.monitoring.enableAxis := TRUE;
   cmJRWinderRearAxisY.monitoring.openBrake := FALSE;
   cmJRWinderRearAxisY.monitoring.jogBackward := FALSE;
   cmJRWinderRearAxisY.monitoring.jogForward := FALSE;
   cmJRWinderRearAxisY.monitoring.moveVelocity := FALSE;
   cmJRWinderRearAxisY.monitoring.stop := FALSE;
   cmJRWinderRearAxisY.monitoring.fastStop := FALSE;
   cmJRWinderRearAxisY.monitoring.torqueLimiting := FALSE;
   cmJRWinderRearAxisY.monitoring.homing := FALSE;
   cmJRWinderRearAxisY.monitoring.posRelative := FALSE;
   cmJRWinderRearAxisY.monitoring.posAbsolute := FALSE;
   cmJRWinderRearAxisY.monitoring.posSuperimposed := FALSE;
   cmJRWinderRearAxisY.monitoring.haltSuperimposed := FALSE;
   cmJRWinderRearAxisY.monitoring.brakeOpened := FALSE;
   cmJRWinderRearAxisY.monitoring.axisEnabled := TRUE;
   cmJRWinderRearAxisY.monitoring.resetActive := FALSE;
   cmJRWinderRearAxisY.monitoring.inVelocity := FALSE;
   cmJRWinderRearAxisY.monitoring.inLimitation := FALSE;
   cmJRWinderRearAxisY.monitoring.inClamping := FALSE;
   cmJRWinderRearAxisY.monitoring.startSync := FALSE;
   cmJRWinderRearAxisY.monitoring.inSync := FALSE;
   cmJRWinderRearAxisY.monitoring.inSimulation := FALSE;
   cmJRWinderRearAxisY.monitoring.jogSelected := FALSE;
   cmJRWinderRearAxisY.monitoring.moveVelocitySelected := FALSE;
   cmJRWinderRearAxisY.monitoring.stopSelected := FALSE;
   cmJRWinderRearAxisY.monitoring.fastStopSelected := FALSE;
   cmJRWinderRearAxisY.monitoring.torqueLimitingSelected := FALSE;
   cmJRWinderRearAxisY.monitoring.homingSelected := FALSE;
   cmJRWinderRearAxisY.monitoring.posRelativeSelected := FALSE;
   cmJRWinderRearAxisY.monitoring.posAbsoluteSelected := FALSE;
   cmJRWinderRearAxisY.monitoring.posSuperimposedSelected := FALSE;
   cmJRWinderRearAxisY.monitoring.haltSuperimposedSelected := FALSE;
   cmJRWinderRearAxisY.monitoring.commandBusy := FALSE;
   cmJRWinderRearAxisY.monitoring.commandDone := FALSE;
   cmJRWinderRearAxisY.monitoring.commandAborted := FALSE;
   cmJRWinderRearAxisY.monitoring.homingCommandBusy := FALSE;
   cmJRWinderRearAxisY.monitoring.homingCommandDone := FALSE;
   cmJRWinderRearAxisY.monitoring.homingCommandAborted := FALSE;
   cmJRWinderRearAxisY.monitoring.superimposedBusy := FALSE;
   cmJRWinderRearAxisY.monitoring.superimposedDone := FALSE;
   cmJRWinderRearAxisY.monitoring.superimposedAborted := FALSE;
   cmJRWinderRearAxisY.monitoring.selectSetPosition := -1;
   cmJRWinderRearAxisY.monitoring.selectionController := FALSE;
   cmJRWinderRearAxisY.monitoring.interlockGeneral := TRUE;
   cmJRWinderRearAxisY.monitoring.interlockJogForward := TRUE;
   cmJRWinderRearAxisY.monitoring.interlockJogBackward := TRUE;
   cmJRWinderRearAxisY.monitoring.interlockWarningGeneral := FALSE;
   cmJRWinderRearAxisY.monitoring.interlockWarningJogForward := FALSE;
   cmJRWinderRearAxisY.monitoring.interlockWarningJogBackward := FALSE;
   cmJRWinderRearAxisY.monitoring.valid := TRUE;
   cmJRWinderRearAxisY.monitoring.busy := TRUE;
   cmJRWinderRearAxisY.monitoring.error := FALSE;
   cmJRWinderRearAxisY.monitoring.status := 16#7002;
   cmJRWinderRearAxisY.monitoring.subfunctionStatus := 16#0000;
   cmJRWinderRearAxisY.monitoring.actualPosition := 0.0;
   cmJRWinderRearAxisY.monitoring.actualSpeed := 0.0;
   cmJRWinderRearAxisY.monitoring.speedUnit := 1062;
   cmJRWinderRearAxisY.monitoring.positionUnit := 1013;
   cmJRWinderRearAxisY.monitoring.axisStatus1 := 16#0200_10E1;
   cmJRWinderRearAxisY.monitoring.axisStatus2 := 16#0000_0000;
   cmJRWinderRearAxisY.monitoring.axisType := 1;
   cmJRWinderRearAxisY.monitoring.maxVelocity := 2500.0;
   cmJRWinderRearAxisY.monitoring.actualCurrent := 0.0;
   cmJRWinderRearAxisY.monitoring.actualTorque := 0.0;
   cmJRWinderRearAxisY.monitoring.velocityOverrideEnabled := FALSE;
   cmJRWinderRearAxisY.monitoring.sinaParaError := FALSE;
   cmJRWinderRearAxisY.monitoring.sinaParaStatus := 16#0000_0000;
   cmJRWinderRearAxisY.configuration.referenceDesignator := WSTRING#'JRWinderRearAxisY';
   cmJRWinderRearAxisY.configuration.disableAlarms := FALSE;
   cmJRWinderRearAxisY.configuration.masterControlPopUp := TRUE;
   cmJRWinderRearAxisY.configuration.setPositions[0].position := 0.0;
   cmJRWinderRearAxisY.configuration.setPositions[1].position := 50.0;
   cmJRWinderRearAxisY.configuration.setPositions[2..15].position := 0.0;
   cmJRWinderRearAxisY.configuration.setPositions[0..1].velocity := 50.0;
   cmJRWinderRearAxisY.configuration.setPositions[2..15].velocity := -1.0;
   cmJRWinderRearAxisY.configuration.setPositions[0..1].acceleration := 500.0;
   cmJRWinderRearAxisY.configuration.setPositions[2..15].acceleration := -1.0;
   cmJRWinderRearAxisY.configuration.setPositions[0..1].deceleration := 500.0;
   cmJRWinderRearAxisY.configuration.setPositions[2..15].deceleration := -1.0;
   cmJRWinderRearAxisY.configuration.setPositions[0..15]."name" := '';
   cmJRWinderFrontAxisY.commandConfiguration.generalSettings.stopOnError := TRUE;
   cmJRWinderFrontAxisY.commandConfiguration.generalSettings.resetWithRestart := FALSE;
   cmJRWinderFrontAxisY.commandConfiguration.generalSettings.abortWaitingSyncCmd := TRUE;
   cmJRWinderFrontAxisY.commandConfiguration.power.startMode := 1;
   cmJRWinderFrontAxisY.commandConfiguration.power.stopMode := 0;
   cmJRWinderFrontAxisY.commandConfiguration.power.syncMotionSimulation := FALSE;
   cmJRWinderFrontAxisY.commandConfiguration.power.syncMotionSimulationExtendedMode := -1;
   cmJRWinderFrontAxisY.commandConfiguration.jog.velocity := 0.0;
   cmJRWinderFrontAxisY.commandConfiguration.jog.acceleration := -1.0;
   cmJRWinderFrontAxisY.commandConfiguration.jog.deceleration := -1.0;
   cmJRWinderFrontAxisY.commandConfiguration.jog.jerk := -1.0;
   cmJRWinderFrontAxisY.commandConfiguration.jog.positionControlled := TRUE;
   cmJRWinderFrontAxisY.commandConfiguration.jog.increment := 0.0;
   cmJRWinderFrontAxisY.commandConfiguration.jog.mode := 0;
   cmJRWinderFrontAxisY.commandConfiguration.moveVelocity.velocity := 0.0;
   cmJRWinderFrontAxisY.commandConfiguration.moveVelocity.acceleration := -1.0;
   cmJRWinderFrontAxisY.commandConfiguration.moveVelocity.deceleration := -1.0;
   cmJRWinderFrontAxisY.commandConfiguration.moveVelocity.jerk := -1.0;
   cmJRWinderFrontAxisY.commandConfiguration.moveVelocity.direction := 0;
   cmJRWinderFrontAxisY.commandConfiguration.moveVelocity.positionControlled := TRUE;
   cmJRWinderFrontAxisY.commandConfiguration.moveVelocity.velocityChangeOnTheFly := FALSE;
   cmJRWinderFrontAxisY.commandConfiguration.stop.deceleration := -1.0;
   cmJRWinderFrontAxisY.commandConfiguration.stop.jerk := -1.0;
   cmJRWinderFrontAxisY.commandConfiguration.stop.abortAcceleration := FALSE;
   cmJRWinderFrontAxisY.commandConfiguration.fastStop.deceleration := -1.0;
   cmJRWinderFrontAxisY.commandConfiguration.fastStop.jerk := -1.0;
   cmJRWinderFrontAxisY.commandConfiguration.fastStop.abortAcceleration := FALSE;
   cmJRWinderFrontAxisY.commandConfiguration.fastStop.replaceStopPossible := FALSE;
   cmJRWinderFrontAxisY.commandConfiguration.torqueLimiting.limit := -1.0;
   cmJRWinderFrontAxisY.commandConfiguration.torqueLimiting.mode := 0;
   cmJRWinderFrontAxisY.commandConfiguration.homing.position := 0.0;
   cmJRWinderFrontAxisY.commandConfiguration.homing.mode := 0;
   cmJRWinderFrontAxisY.commandConfiguration.homing.sensor := 0;
   cmJRWinderFrontAxisY.commandConfiguration.homing.extendedMode := -1;
   cmJRWinderFrontAxisY.commandConfiguration.homing.extendedModeTorqueLimit := 0.0;
   cmJRWinderFrontAxisY.commandConfiguration.homing.extendedModeTargetPosition := 0.0;
   cmJRWinderFrontAxisY.commandConfiguration.posRelative.distance := 0.0;
   cmJRWinderFrontAxisY.commandConfiguration.posRelative.velocity := -1.0;
   cmJRWinderFrontAxisY.commandConfiguration.posRelative.acceleration := -1.0;
   cmJRWinderFrontAxisY.commandConfiguration.posRelative.deceleration := -1.0;
   cmJRWinderFrontAxisY.commandConfiguration.posRelative.jerk := -1.0;
   cmJRWinderFrontAxisY.commandConfiguration.posRelative.direction := 0;
   cmJRWinderFrontAxisY.commandConfiguration.posAbsolute.position := -22.0;
   cmJRWinderFrontAxisY.commandConfiguration.posAbsolute.velocity := 30.0;
   cmJRWinderFrontAxisY.commandConfiguration.posAbsolute.acceleration := 30.0;
   cmJRWinderFrontAxisY.commandConfiguration.posAbsolute.deceleration := 30.0;
   cmJRWinderFrontAxisY.commandConfiguration.posAbsolute.jerk := -1.0;
   cmJRWinderFrontAxisY.commandConfiguration.posAbsolute.direction := 1;
   cmJRWinderFrontAxisY.commandConfiguration.posAbsolute.positionChangeOnTheFly := FALSE;
   cmJRWinderFrontAxisY.commandConfiguration.posAbsolute.velocityChangeOnTheFly := FALSE;
   cmJRWinderFrontAxisY.commandConfiguration.posSuperimposed.distance := 0.0;
   cmJRWinderFrontAxisY.commandConfiguration.posSuperimposed.velocityDiff := -1.0;
   cmJRWinderFrontAxisY.commandConfiguration.posSuperimposed.acceleration := -1.0;
   cmJRWinderFrontAxisY.commandConfiguration.posSuperimposed.deceleration := -1.0;
   cmJRWinderFrontAxisY.commandConfiguration.posSuperimposed.jerk := -1.0;
   cmJRWinderFrontAxisY.commandConfiguration.posSuperimposed.direction := 0;
   cmJRWinderFrontAxisY.commandConfiguration.haltSuperimposed.deceleration := -1.0;
   cmJRWinderFrontAxisY.commandConfiguration.haltSuperimposed.jerk := -1.0;
   cmJRWinderFrontAxisY.commandConfiguration.haltSuperimposed.abortAcceleration := FALSE;
   cmJRWinderFrontAxisY.commandConfiguration.gearInRelative.ratioNumerator := 1;
   cmJRWinderFrontAxisY.commandConfiguration.gearInRelative.ratioDenominator := 1;
   cmJRWinderFrontAxisY.commandConfiguration.gearInRelative.acceleration := -1.0;
   cmJRWinderFrontAxisY.commandConfiguration.gearInRelative.deceleration := -1.0;
   cmJRWinderFrontAxisY.commandConfiguration.gearInRelative.jerk := -1.0;
   cmJRWinderFrontAxisY.commandConfiguration.gearInRelative.ratioChangeOnTheFly := FALSE;
   cmJRWinderFrontAxisY.commandConfiguration.gearInAbsolute.ratioNumerator := 1;
   cmJRWinderFrontAxisY.commandConfiguration.gearInAbsolute.ratioDenominator := 1;
   cmJRWinderFrontAxisY.commandConfiguration.gearInAbsolute.masterSyncPosition := 0.0;
   cmJRWinderFrontAxisY.commandConfiguration.gearInAbsolute.slaveSyncPosition := 0.0;
   cmJRWinderFrontAxisY.commandConfiguration.gearInAbsolute.syncProfileReference := 1;
   cmJRWinderFrontAxisY.commandConfiguration.gearInAbsolute.masterStartDistance := 0.0;
   cmJRWinderFrontAxisY.commandConfiguration.gearInAbsolute.velocity := -1.0;
   cmJRWinderFrontAxisY.commandConfiguration.gearInAbsolute.acceleration := -1.0;
   cmJRWinderFrontAxisY.commandConfiguration.gearInAbsolute.deceleration := -1.0;
   cmJRWinderFrontAxisY.commandConfiguration.gearInAbsolute.jerk := -1.0;
   cmJRWinderFrontAxisY.commandConfiguration.gearInAbsolute.syncDirection := 1;
   cmJRWinderFrontAxisY.commandConfiguration.gearInAbsolute.ratioChangeOnTheFly := FALSE;
   cmJRWinderFrontAxisY.commandConfiguration.gearInVelocity.continuousUpdate := FALSE;
   cmJRWinderFrontAxisY.commandConfiguration.gearInVelocity.ratioNumerator := 1;
   cmJRWinderFrontAxisY.commandConfiguration.gearInVelocity.ratioDenominator := 1;
   cmJRWinderFrontAxisY.commandConfiguration.gearInVelocity.acceleration := -1.0;
   cmJRWinderFrontAxisY.commandConfiguration.gearInVelocity.deceleration := -1.0;
   cmJRWinderFrontAxisY.commandConfiguration.gearInVelocity.jerk := -1.0;
   cmJRWinderFrontAxisY.commandConfiguration.gearInVelocity.positionControlled := FALSE;
   cmJRWinderFrontAxisY.commandConfiguration.camIn.masterOffset := 0.0;
   cmJRWinderFrontAxisY.commandConfiguration.camIn.slaveOffset := 0.0;
   cmJRWinderFrontAxisY.commandConfiguration.camIn.masterScaling := 1.0;
   cmJRWinderFrontAxisY.commandConfiguration.camIn.slaveScaling := 1.0;
   cmJRWinderFrontAxisY.commandConfiguration.camIn.masterSyncPosition := 0.0;
   cmJRWinderFrontAxisY.commandConfiguration.camIn.syncProfileReference := 1;
   cmJRWinderFrontAxisY.commandConfiguration.camIn.masterStartDistance := 0.0;
   cmJRWinderFrontAxisY.commandConfiguration.camIn.velocity := -1.0;
   cmJRWinderFrontAxisY.commandConfiguration.camIn.acceleration := -1.0;
   cmJRWinderFrontAxisY.commandConfiguration.camIn.deceleration := -1.0;
   cmJRWinderFrontAxisY.commandConfiguration.camIn.jerk := -1.0;
   cmJRWinderFrontAxisY.commandConfiguration.camIn.applicationMode := 0;
   cmJRWinderFrontAxisY.commandConfiguration.camIn.syncDirection := 1;
   cmJRWinderFrontAxisY.commandConfiguration.gearOutCamOut.slavePosition := 0.0;
   cmJRWinderFrontAxisY.commandConfiguration.gearOutCamOut.syncProfileReference := 1;
   cmJRWinderFrontAxisY.commandConfiguration.gearOutCamOut.masterStopDistance := 0.0;
   cmJRWinderFrontAxisY.commandConfiguration.gearOutCamOut.deceleration := -1.0;
   cmJRWinderFrontAxisY.commandConfiguration.gearOutCamOut.jerk := -1.0;
   cmJRWinderFrontAxisY.commandConfiguration.gearOutCamOut.syncOutDirection := 3;
   cmJRWinderFrontAxisY.commandConfiguration.gearOutCamOut.gearOutCamOutMode := -1;
   cmJRWinderFrontAxisY.commandConfiguration.phasing.phaseShift := 0.0;
   cmJRWinderFrontAxisY.commandConfiguration.phasing.velocity := -1.0;
   cmJRWinderFrontAxisY.commandConfiguration.phasing.acceleration := -1.0;
   cmJRWinderFrontAxisY.commandConfiguration.phasing.deceleration := -1.0;
   cmJRWinderFrontAxisY.commandConfiguration.phasing.jerk := -1.0;
   cmJRWinderFrontAxisY.commandConfiguration.phasing.profileReference := 0;
   cmJRWinderFrontAxisY.commandConfiguration.phasing.phasingDistance := 0.0;
   cmJRWinderFrontAxisY.commandConfiguration.phasing.startPosition := 0.0;
   cmJRWinderFrontAxisY.commandConfiguration.phasing.direction := 3;
   cmJRWinderFrontAxisY.commandConfiguration.phasing.phaseAbsolute := TRUE;
   cmJRWinderFrontAxisY.commandConfiguration.phasing.phaseShiftChangeOnTheFly := FALSE;
   cmJRWinderFrontAxisY.commandConfiguration.offset.offset := 0.0;
   cmJRWinderFrontAxisY.commandConfiguration.offset.profileReference := 1;
   cmJRWinderFrontAxisY.commandConfiguration.offset.offsetDistance := 0.0;
   cmJRWinderFrontAxisY.commandConfiguration.offset.startPosition := 0.0;
   cmJRWinderFrontAxisY.commandConfiguration.offset.direction := 3;
   cmJRWinderFrontAxisY.commandConfiguration.offset.offsetAbsolute := TRUE;
   cmJRWinderFrontAxisY.commandConfiguration.offset.offsetChangeOnTheFly := FALSE;
   cmJRWinderFrontAxisY.commands.enableMasterControl := TRUE;
   cmJRWinderFrontAxisY.commands.enableAxis := FALSE;
   cmJRWinderFrontAxisY.commands.resetAxis := FALSE;
   cmJRWinderFrontAxisY.commands.openBrake := FALSE;
   cmJRWinderFrontAxisY.commands.jogForward := FALSE;
   cmJRWinderFrontAxisY.commands.jogBackward := FALSE;
   cmJRWinderFrontAxisY.commands.moveVelocity := FALSE;
   cmJRWinderFrontAxisY.commands.stop := FALSE;
   cmJRWinderFrontAxisY.commands.fastStop := FALSE;
   cmJRWinderFrontAxisY.commands.torqueLimiting := FALSE;
   cmJRWinderFrontAxisY.commands.homing := FALSE;
   cmJRWinderFrontAxisY.commands.posRelative := FALSE;
   cmJRWinderFrontAxisY.commands.posAbsolute := FALSE;
   cmJRWinderFrontAxisY.commands.posSuperimposed := FALSE;
   cmJRWinderFrontAxisY.commands.haltSuperimposed := FALSE;
   cmJRWinderFrontAxisY.commands.selectSetPosition := -1;
   cmJRWinderFrontAxisY.commands.uploadParameters := FALSE;
   cmJRWinderFrontAxisY.commands.refreshConfiguration := FALSE;
   cmJRWinderFrontAxisY.commands.editConfiguration := FALSE;
   cmJRWinderFrontAxisY.commands.saveConfiguration := FALSE;
   cmJRWinderFrontAxisY.commands.uploadCurrentTorque := FALSE;
   cmJRWinderFrontAxisY.commands.reset := FALSE;
   cmJRWinderFrontAxisY.monitoring.enable := TRUE;
   cmJRWinderFrontAxisY.monitoring.referenceDesignator := WSTRING#'JRWinderFrontAxisY';
   cmJRWinderFrontAxisY.monitoring.enabled := TRUE;
   cmJRWinderFrontAxisY.monitoring.enableManualCmds := FALSE;
   cmJRWinderFrontAxisY.monitoring.reset := FALSE;
   cmJRWinderFrontAxisY.monitoring.resetAxis := FALSE;
   cmJRWinderFrontAxisY.monitoring.enableAxis := TRUE;
   cmJRWinderFrontAxisY.monitoring.openBrake := FALSE;
   cmJRWinderFrontAxisY.monitoring.jogBackward := FALSE;
   cmJRWinderFrontAxisY.monitoring.jogForward := FALSE;
   cmJRWinderFrontAxisY.monitoring.moveVelocity := FALSE;
   cmJRWinderFrontAxisY.monitoring.stop := FALSE;
   cmJRWinderFrontAxisY.monitoring.fastStop := FALSE;
   cmJRWinderFrontAxisY.monitoring.torqueLimiting := FALSE;
   cmJRWinderFrontAxisY.monitoring.homing := FALSE;
   cmJRWinderFrontAxisY.monitoring.posRelative := FALSE;
   cmJRWinderFrontAxisY.monitoring.posAbsolute := FALSE;
   cmJRWinderFrontAxisY.monitoring.posSuperimposed := FALSE;
   cmJRWinderFrontAxisY.monitoring.haltSuperimposed := FALSE;
   cmJRWinderFrontAxisY.monitoring.brakeOpened := FALSE;
   cmJRWinderFrontAxisY.monitoring.axisEnabled := TRUE;
   cmJRWinderFrontAxisY.monitoring.resetActive := FALSE;
   cmJRWinderFrontAxisY.monitoring.inVelocity := FALSE;
   cmJRWinderFrontAxisY.monitoring.inLimitation := FALSE;
   cmJRWinderFrontAxisY.monitoring.inClamping := FALSE;
   cmJRWinderFrontAxisY.monitoring.startSync := FALSE;
   cmJRWinderFrontAxisY.monitoring.inSync := FALSE;
   cmJRWinderFrontAxisY.monitoring.inSimulation := FALSE;
   cmJRWinderFrontAxisY.monitoring.jogSelected := FALSE;
   cmJRWinderFrontAxisY.monitoring.moveVelocitySelected := FALSE;
   cmJRWinderFrontAxisY.monitoring.stopSelected := FALSE;
   cmJRWinderFrontAxisY.monitoring.fastStopSelected := FALSE;
   cmJRWinderFrontAxisY.monitoring.torqueLimitingSelected := FALSE;
   cmJRWinderFrontAxisY.monitoring.homingSelected := FALSE;
   cmJRWinderFrontAxisY.monitoring.posRelativeSelected := FALSE;
   cmJRWinderFrontAxisY.monitoring.posAbsoluteSelected := FALSE;
   cmJRWinderFrontAxisY.monitoring.posSuperimposedSelected := FALSE;
   cmJRWinderFrontAxisY.monitoring.haltSuperimposedSelected := FALSE;
   cmJRWinderFrontAxisY.monitoring.commandBusy := FALSE;
   cmJRWinderFrontAxisY.monitoring.commandDone := FALSE;
   cmJRWinderFrontAxisY.monitoring.commandAborted := FALSE;
   cmJRWinderFrontAxisY.monitoring.homingCommandBusy := FALSE;
   cmJRWinderFrontAxisY.monitoring.homingCommandDone := FALSE;
   cmJRWinderFrontAxisY.monitoring.homingCommandAborted := FALSE;
   cmJRWinderFrontAxisY.monitoring.superimposedBusy := FALSE;
   cmJRWinderFrontAxisY.monitoring.superimposedDone := FALSE;
   cmJRWinderFrontAxisY.monitoring.superimposedAborted := FALSE;
   cmJRWinderFrontAxisY.monitoring.selectSetPosition := -1;
   cmJRWinderFrontAxisY.monitoring.selectionController := FALSE;
   cmJRWinderFrontAxisY.monitoring.interlockGeneral := TRUE;
   cmJRWinderFrontAxisY.monitoring.interlockJogForward := TRUE;
   cmJRWinderFrontAxisY.monitoring.interlockJogBackward := TRUE;
   cmJRWinderFrontAxisY.monitoring.interlockWarningGeneral := FALSE;
   cmJRWinderFrontAxisY.monitoring.interlockWarningJogForward := FALSE;
   cmJRWinderFrontAxisY.monitoring.interlockWarningJogBackward := FALSE;
   cmJRWinderFrontAxisY.monitoring.valid := TRUE;
   cmJRWinderFrontAxisY.monitoring.busy := TRUE;
   cmJRWinderFrontAxisY.monitoring.error := FALSE;
   cmJRWinderFrontAxisY.monitoring.status := 16#7002;
   cmJRWinderFrontAxisY.monitoring.subfunctionStatus := 16#0000;
   cmJRWinderFrontAxisY.monitoring.actualPosition := 0.0;
   cmJRWinderFrontAxisY.monitoring.actualSpeed := 0.0;
   cmJRWinderFrontAxisY.monitoring.speedUnit := 1062;
   cmJRWinderFrontAxisY.monitoring.positionUnit := 1013;
   cmJRWinderFrontAxisY.monitoring.axisStatus1 := 16#0200_10E1;
   cmJRWinderFrontAxisY.monitoring.axisStatus2 := 16#0000_0000;
   cmJRWinderFrontAxisY.monitoring.axisType := 1;
   cmJRWinderFrontAxisY.monitoring.maxVelocity := 2500.0;
   cmJRWinderFrontAxisY.monitoring.actualCurrent := 0.0;
   cmJRWinderFrontAxisY.monitoring.actualTorque := 0.0;
   cmJRWinderFrontAxisY.monitoring.velocityOverrideEnabled := FALSE;
   cmJRWinderFrontAxisY.monitoring.sinaParaError := FALSE;
   cmJRWinderFrontAxisY.monitoring.sinaParaStatus := 16#0000_0000;
   cmJRWinderFrontAxisY.configuration.referenceDesignator := WSTRING#'JRWinderFrontAxisY';
   cmJRWinderFrontAxisY.configuration.disableAlarms := FALSE;
   cmJRWinderFrontAxisY.configuration.masterControlPopUp := TRUE;
   cmJRWinderFrontAxisY.configuration.setPositions[0].position := 0.0;
   cmJRWinderFrontAxisY.configuration.setPositions[1].position := 50.0;
   cmJRWinderFrontAxisY.configuration.setPositions[2..15].position := 0.0;
   cmJRWinderFrontAxisY.configuration.setPositions[0..1].velocity := 50.0;
   cmJRWinderFrontAxisY.configuration.setPositions[2..15].velocity := -1.0;
   cmJRWinderFrontAxisY.configuration.setPositions[0..1].acceleration := 500.0;
   cmJRWinderFrontAxisY.configuration.setPositions[2..15].acceleration := -1.0;
   cmJRWinderFrontAxisY.configuration.setPositions[0..1].deceleration := 500.0;
   cmJRWinderFrontAxisY.configuration.setPositions[2..15].deceleration := -1.0;
   cmJRWinderFrontAxisY.configuration.setPositions[0..15]."name" := '';
   cmJRWinderAxisB.commandConfiguration.generalSettings.stopOnError := TRUE;
   cmJRWinderAxisB.commandConfiguration.generalSettings.resetWithRestart := FALSE;
   cmJRWinderAxisB.commandConfiguration.generalSettings.abortWaitingSyncCmd := TRUE;
   cmJRWinderAxisB.commandConfiguration.power.startMode := 1;
   cmJRWinderAxisB.commandConfiguration.power.stopMode := 0;
   cmJRWinderAxisB.commandConfiguration.power.syncMotionSimulation := FALSE;
   cmJRWinderAxisB.commandConfiguration.power.syncMotionSimulationExtendedMode := -1;
   cmJRWinderAxisB.commandConfiguration.jog.velocity := 0.0;
   cmJRWinderAxisB.commandConfiguration.jog.acceleration := -1.0;
   cmJRWinderAxisB.commandConfiguration.jog.deceleration := -1.0;
   cmJRWinderAxisB.commandConfiguration.jog.jerk := -1.0;
   cmJRWinderAxisB.commandConfiguration.jog.positionControlled := TRUE;
   cmJRWinderAxisB.commandConfiguration.jog.increment := 0.0;
   cmJRWinderAxisB.commandConfiguration.jog.mode := 0;
   cmJRWinderAxisB.commandConfiguration.moveVelocity.velocity := 0.0;
   cmJRWinderAxisB.commandConfiguration.moveVelocity.acceleration := -1.0;
   cmJRWinderAxisB.commandConfiguration.moveVelocity.deceleration := -1.0;
   cmJRWinderAxisB.commandConfiguration.moveVelocity.jerk := -1.0;
   cmJRWinderAxisB.commandConfiguration.moveVelocity.direction := 0;
   cmJRWinderAxisB.commandConfiguration.moveVelocity.positionControlled := TRUE;
   cmJRWinderAxisB.commandConfiguration.moveVelocity.velocityChangeOnTheFly := FALSE;
   cmJRWinderAxisB.commandConfiguration.stop.deceleration := -1.0;
   cmJRWinderAxisB.commandConfiguration.stop.jerk := -1.0;
   cmJRWinderAxisB.commandConfiguration.stop.abortAcceleration := FALSE;
   cmJRWinderAxisB.commandConfiguration.fastStop.deceleration := -1.0;
   cmJRWinderAxisB.commandConfiguration.fastStop.jerk := -1.0;
   cmJRWinderAxisB.commandConfiguration.fastStop.abortAcceleration := FALSE;
   cmJRWinderAxisB.commandConfiguration.fastStop.replaceStopPossible := FALSE;
   cmJRWinderAxisB.commandConfiguration.torqueLimiting.limit := -1.0;
   cmJRWinderAxisB.commandConfiguration.torqueLimiting.mode := 0;
   cmJRWinderAxisB.commandConfiguration.homing.position := 0.0;
   cmJRWinderAxisB.commandConfiguration.homing.mode := 0;
   cmJRWinderAxisB.commandConfiguration.homing.sensor := 0;
   cmJRWinderAxisB.commandConfiguration.homing.extendedMode := -1;
   cmJRWinderAxisB.commandConfiguration.homing.extendedModeTorqueLimit := 0.0;
   cmJRWinderAxisB.commandConfiguration.homing.extendedModeTargetPosition := 0.0;
   cmJRWinderAxisB.commandConfiguration.posRelative.distance := 0.0;
   cmJRWinderAxisB.commandConfiguration.posRelative.velocity := 10.0;
   cmJRWinderAxisB.commandConfiguration.posRelative.acceleration := 30.0;
   cmJRWinderAxisB.commandConfiguration.posRelative.deceleration := 30.0;
   cmJRWinderAxisB.commandConfiguration.posRelative.jerk := -1.0;
   cmJRWinderAxisB.commandConfiguration.posRelative.direction := 0;
   cmJRWinderAxisB.commandConfiguration.posAbsolute.position := 0.0;
   cmJRWinderAxisB.commandConfiguration.posAbsolute.velocity := -1.0;
   cmJRWinderAxisB.commandConfiguration.posAbsolute.acceleration := -1.0;
   cmJRWinderAxisB.commandConfiguration.posAbsolute.deceleration := -1.0;
   cmJRWinderAxisB.commandConfiguration.posAbsolute.jerk := -1.0;
   cmJRWinderAxisB.commandConfiguration.posAbsolute.direction := 1;
   cmJRWinderAxisB.commandConfiguration.posAbsolute.positionChangeOnTheFly := FALSE;
   cmJRWinderAxisB.commandConfiguration.posAbsolute.velocityChangeOnTheFly := FALSE;
   cmJRWinderAxisB.commandConfiguration.posSuperimposed.distance := 0.0;
   cmJRWinderAxisB.commandConfiguration.posSuperimposed.velocityDiff := -1.0;
   cmJRWinderAxisB.commandConfiguration.posSuperimposed.acceleration := -1.0;
   cmJRWinderAxisB.commandConfiguration.posSuperimposed.deceleration := -1.0;
   cmJRWinderAxisB.commandConfiguration.posSuperimposed.jerk := -1.0;
   cmJRWinderAxisB.commandConfiguration.posSuperimposed.direction := 0;
   cmJRWinderAxisB.commandConfiguration.haltSuperimposed.deceleration := -1.0;
   cmJRWinderAxisB.commandConfiguration.haltSuperimposed.jerk := -1.0;
   cmJRWinderAxisB.commandConfiguration.haltSuperimposed.abortAcceleration := FALSE;
   cmJRWinderAxisB.commandConfiguration.gearInRelative.ratioNumerator := 1;
   cmJRWinderAxisB.commandConfiguration.gearInRelative.ratioDenominator := 1;
   cmJRWinderAxisB.commandConfiguration.gearInRelative.acceleration := -1.0;
   cmJRWinderAxisB.commandConfiguration.gearInRelative.deceleration := -1.0;
   cmJRWinderAxisB.commandConfiguration.gearInRelative.jerk := -1.0;
   cmJRWinderAxisB.commandConfiguration.gearInRelative.ratioChangeOnTheFly := FALSE;
   cmJRWinderAxisB.commandConfiguration.gearInAbsolute.ratioNumerator := 1;
   cmJRWinderAxisB.commandConfiguration.gearInAbsolute.ratioDenominator := 1;
   cmJRWinderAxisB.commandConfiguration.gearInAbsolute.masterSyncPosition := 0.0;
   cmJRWinderAxisB.commandConfiguration.gearInAbsolute.slaveSyncPosition := 0.0;
   cmJRWinderAxisB.commandConfiguration.gearInAbsolute.syncProfileReference := 1;
   cmJRWinderAxisB.commandConfiguration.gearInAbsolute.masterStartDistance := 0.0;
   cmJRWinderAxisB.commandConfiguration.gearInAbsolute.velocity := -1.0;
   cmJRWinderAxisB.commandConfiguration.gearInAbsolute.acceleration := -1.0;
   cmJRWinderAxisB.commandConfiguration.gearInAbsolute.deceleration := -1.0;
   cmJRWinderAxisB.commandConfiguration.gearInAbsolute.jerk := -1.0;
   cmJRWinderAxisB.commandConfiguration.gearInAbsolute.syncDirection := 1;
   cmJRWinderAxisB.commandConfiguration.gearInAbsolute.ratioChangeOnTheFly := FALSE;
   cmJRWinderAxisB.commandConfiguration.gearInVelocity.continuousUpdate := FALSE;
   cmJRWinderAxisB.commandConfiguration.gearInVelocity.ratioNumerator := 1;
   cmJRWinderAxisB.commandConfiguration.gearInVelocity.ratioDenominator := 1;
   cmJRWinderAxisB.commandConfiguration.gearInVelocity.acceleration := -1.0;
   cmJRWinderAxisB.commandConfiguration.gearInVelocity.deceleration := -1.0;
   cmJRWinderAxisB.commandConfiguration.gearInVelocity.jerk := -1.0;
   cmJRWinderAxisB.commandConfiguration.gearInVelocity.positionControlled := FALSE;
   cmJRWinderAxisB.commandConfiguration.camIn.masterOffset := 0.0;
   cmJRWinderAxisB.commandConfiguration.camIn.slaveOffset := 0.0;
   cmJRWinderAxisB.commandConfiguration.camIn.masterScaling := 1.0;
   cmJRWinderAxisB.commandConfiguration.camIn.slaveScaling := 1.0;
   cmJRWinderAxisB.commandConfiguration.camIn.masterSyncPosition := 0.0;
   cmJRWinderAxisB.commandConfiguration.camIn.syncProfileReference := 1;
   cmJRWinderAxisB.commandConfiguration.camIn.masterStartDistance := 0.0;
   cmJRWinderAxisB.commandConfiguration.camIn.velocity := -1.0;
   cmJRWinderAxisB.commandConfiguration.camIn.acceleration := -1.0;
   cmJRWinderAxisB.commandConfiguration.camIn.deceleration := -1.0;
   cmJRWinderAxisB.commandConfiguration.camIn.jerk := -1.0;
   cmJRWinderAxisB.commandConfiguration.camIn.applicationMode := 0;
   cmJRWinderAxisB.commandConfiguration.camIn.syncDirection := 1;
   cmJRWinderAxisB.commandConfiguration.gearOutCamOut.slavePosition := 0.0;
   cmJRWinderAxisB.commandConfiguration.gearOutCamOut.syncProfileReference := 1;
   cmJRWinderAxisB.commandConfiguration.gearOutCamOut.masterStopDistance := 0.0;
   cmJRWinderAxisB.commandConfiguration.gearOutCamOut.deceleration := -1.0;
   cmJRWinderAxisB.commandConfiguration.gearOutCamOut.jerk := -1.0;
   cmJRWinderAxisB.commandConfiguration.gearOutCamOut.syncOutDirection := 3;
   cmJRWinderAxisB.commandConfiguration.gearOutCamOut.gearOutCamOutMode := -1;
   cmJRWinderAxisB.commandConfiguration.phasing.phaseShift := 0.0;
   cmJRWinderAxisB.commandConfiguration.phasing.velocity := -1.0;
   cmJRWinderAxisB.commandConfiguration.phasing.acceleration := -1.0;
   cmJRWinderAxisB.commandConfiguration.phasing.deceleration := -1.0;
   cmJRWinderAxisB.commandConfiguration.phasing.jerk := -1.0;
   cmJRWinderAxisB.commandConfiguration.phasing.profileReference := 0;
   cmJRWinderAxisB.commandConfiguration.phasing.phasingDistance := 0.0;
   cmJRWinderAxisB.commandConfiguration.phasing.startPosition := 0.0;
   cmJRWinderAxisB.commandConfiguration.phasing.direction := 3;
   cmJRWinderAxisB.commandConfiguration.phasing.phaseAbsolute := TRUE;
   cmJRWinderAxisB.commandConfiguration.phasing.phaseShiftChangeOnTheFly := FALSE;
   cmJRWinderAxisB.commandConfiguration.offset.offset := 0.0;
   cmJRWinderAxisB.commandConfiguration.offset.profileReference := 1;
   cmJRWinderAxisB.commandConfiguration.offset.offsetDistance := 0.0;
   cmJRWinderAxisB.commandConfiguration.offset.startPosition := 0.0;
   cmJRWinderAxisB.commandConfiguration.offset.direction := 3;
   cmJRWinderAxisB.commandConfiguration.offset.offsetAbsolute := TRUE;
   cmJRWinderAxisB.commandConfiguration.offset.offsetChangeOnTheFly := FALSE;
   cmJRWinderAxisB.commands.enableMasterControl := TRUE;
   cmJRWinderAxisB.commands.enableAxis := FALSE;
   cmJRWinderAxisB.commands.resetAxis := FALSE;
   cmJRWinderAxisB.commands.openBrake := FALSE;
   cmJRWinderAxisB.commands.jogForward := FALSE;
   cmJRWinderAxisB.commands.jogBackward := FALSE;
   cmJRWinderAxisB.commands.moveVelocity := FALSE;
   cmJRWinderAxisB.commands.stop := FALSE;
   cmJRWinderAxisB.commands.fastStop := FALSE;
   cmJRWinderAxisB.commands.torqueLimiting := FALSE;
   cmJRWinderAxisB.commands.homing := FALSE;
   cmJRWinderAxisB.commands.posRelative := FALSE;
   cmJRWinderAxisB.commands.posAbsolute := FALSE;
   cmJRWinderAxisB.commands.posSuperimposed := FALSE;
   cmJRWinderAxisB.commands.haltSuperimposed := FALSE;
   cmJRWinderAxisB.commands.selectSetPosition := -1;
   cmJRWinderAxisB.commands.uploadParameters := FALSE;
   cmJRWinderAxisB.commands.refreshConfiguration := FALSE;
   cmJRWinderAxisB.commands.editConfiguration := FALSE;
   cmJRWinderAxisB.commands.saveConfiguration := FALSE;
   cmJRWinderAxisB.commands.uploadCurrentTorque := FALSE;
   cmJRWinderAxisB.commands.reset := FALSE;
   cmJRWinderAxisB.monitoring.enable := TRUE;
   cmJRWinderAxisB.monitoring.referenceDesignator := WSTRING#'JRWinderAxisB';
   cmJRWinderAxisB.monitoring.enabled := TRUE;
   cmJRWinderAxisB.monitoring.enableManualCmds := FALSE;
   cmJRWinderAxisB.monitoring.reset := FALSE;
   cmJRWinderAxisB.monitoring.resetAxis := FALSE;
   cmJRWinderAxisB.monitoring.enableAxis := TRUE;
   cmJRWinderAxisB.monitoring.openBrake := FALSE;
   cmJRWinderAxisB.monitoring.jogBackward := FALSE;
   cmJRWinderAxisB.monitoring.jogForward := FALSE;
   cmJRWinderAxisB.monitoring.moveVelocity := FALSE;
   cmJRWinderAxisB.monitoring.stop := FALSE;
   cmJRWinderAxisB.monitoring.fastStop := FALSE;
   cmJRWinderAxisB.monitoring.torqueLimiting := FALSE;
   cmJRWinderAxisB.monitoring.homing := FALSE;
   cmJRWinderAxisB.monitoring.posRelative := FALSE;
   cmJRWinderAxisB.monitoring.posAbsolute := FALSE;
   cmJRWinderAxisB.monitoring.posSuperimposed := FALSE;
   cmJRWinderAxisB.monitoring.haltSuperimposed := FALSE;
   cmJRWinderAxisB.monitoring.brakeOpened := FALSE;
   cmJRWinderAxisB.monitoring.axisEnabled := TRUE;
   cmJRWinderAxisB.monitoring.resetActive := FALSE;
   cmJRWinderAxisB.monitoring.inVelocity := FALSE;
   cmJRWinderAxisB.monitoring.inLimitation := FALSE;
   cmJRWinderAxisB.monitoring.inClamping := FALSE;
   cmJRWinderAxisB.monitoring.startSync := FALSE;
   cmJRWinderAxisB.monitoring.inSync := FALSE;
   cmJRWinderAxisB.monitoring.inSimulation := FALSE;
   cmJRWinderAxisB.monitoring.jogSelected := FALSE;
   cmJRWinderAxisB.monitoring.moveVelocitySelected := FALSE;
   cmJRWinderAxisB.monitoring.stopSelected := FALSE;
   cmJRWinderAxisB.monitoring.fastStopSelected := FALSE;
   cmJRWinderAxisB.monitoring.torqueLimitingSelected := FALSE;
   cmJRWinderAxisB.monitoring.homingSelected := FALSE;
   cmJRWinderAxisB.monitoring.posRelativeSelected := FALSE;
   cmJRWinderAxisB.monitoring.posAbsoluteSelected := FALSE;
   cmJRWinderAxisB.monitoring.posSuperimposedSelected := FALSE;
   cmJRWinderAxisB.monitoring.haltSuperimposedSelected := FALSE;
   cmJRWinderAxisB.monitoring.commandBusy := FALSE;
   cmJRWinderAxisB.monitoring.commandDone := FALSE;
   cmJRWinderAxisB.monitoring.commandAborted := FALSE;
   cmJRWinderAxisB.monitoring.homingCommandBusy := FALSE;
   cmJRWinderAxisB.monitoring.homingCommandDone := FALSE;
   cmJRWinderAxisB.monitoring.homingCommandAborted := FALSE;
   cmJRWinderAxisB.monitoring.superimposedBusy := FALSE;
   cmJRWinderAxisB.monitoring.superimposedDone := FALSE;
   cmJRWinderAxisB.monitoring.superimposedAborted := FALSE;
   cmJRWinderAxisB.monitoring.selectSetPosition := -1;
   cmJRWinderAxisB.monitoring.selectionController := FALSE;
   cmJRWinderAxisB.monitoring.interlockGeneral := TRUE;
   cmJRWinderAxisB.monitoring.interlockJogForward := TRUE;
   cmJRWinderAxisB.monitoring.interlockJogBackward := TRUE;
   cmJRWinderAxisB.monitoring.interlockWarningGeneral := FALSE;
   cmJRWinderAxisB.monitoring.interlockWarningJogForward := FALSE;
   cmJRWinderAxisB.monitoring.interlockWarningJogBackward := FALSE;
   cmJRWinderAxisB.monitoring.valid := TRUE;
   cmJRWinderAxisB.monitoring.busy := TRUE;
   cmJRWinderAxisB.monitoring.error := FALSE;
   cmJRWinderAxisB.monitoring.status := 16#7002;
   cmJRWinderAxisB.monitoring.subfunctionStatus := 16#0000;
   cmJRWinderAxisB.monitoring.actualPosition := 0.0;
   cmJRWinderAxisB.monitoring.actualSpeed := 0.0;
   cmJRWinderAxisB.monitoring.speedUnit := 1521;
   cmJRWinderAxisB.monitoring.positionUnit := 1005;
   cmJRWinderAxisB.monitoring.axisStatus1 := 16#0200_10E1;
   cmJRWinderAxisB.monitoring.axisStatus2 := 16#0000_0000;
   cmJRWinderAxisB.monitoring.axisType := 1;
   cmJRWinderAxisB.monitoring.maxVelocity := 18000.0;
   cmJRWinderAxisB.monitoring.actualCurrent := 0.0;
   cmJRWinderAxisB.monitoring.actualTorque := 0.0;
   cmJRWinderAxisB.monitoring.velocityOverrideEnabled := FALSE;
   cmJRWinderAxisB.monitoring.sinaParaError := FALSE;
   cmJRWinderAxisB.monitoring.sinaParaStatus := 16#0000_0000;
   cmJRWinderAxisB.configuration.referenceDesignator := WSTRING#'JRWinderAxisB';
   cmJRWinderAxisB.configuration.disableAlarms := FALSE;
   cmJRWinderAxisB.configuration.masterControlPopUp := TRUE;
   cmJRWinderAxisB.configuration.setPositions[0].position := 0.0;
   cmJRWinderAxisB.configuration.setPositions[1].position := 360.0;
   cmJRWinderAxisB.configuration.setPositions[2].position := 450.0;
   cmJRWinderAxisB.configuration.setPositions[3].position := 540.0;
   cmJRWinderAxisB.configuration.setPositions[4..15].position := 0.0;
   cmJRWinderAxisB.configuration.setPositions[0..3].velocity := 100.0;
   cmJRWinderAxisB.configuration.setPositions[4..15].velocity := -1.0;
   cmJRWinderAxisB.configuration.setPositions[0..3].acceleration := 1000.0;
   cmJRWinderAxisB.configuration.setPositions[4..15].acceleration := -1.0;
   cmJRWinderAxisB.configuration.setPositions[0..3].deceleration := 1000.0;
   cmJRWinderAxisB.configuration.setPositions[4..15].deceleration := -1.0;
   cmJRWinderAxisB.configuration.setPositions[0..15]."name" := '';
   cmJRPusherAxisZ.commandConfiguration.generalSettings.stopOnError := TRUE;
   cmJRPusherAxisZ.commandConfiguration.generalSettings.resetWithRestart := FALSE;
   cmJRPusherAxisZ.commandConfiguration.generalSettings.abortWaitingSyncCmd := TRUE;
   cmJRPusherAxisZ.commandConfiguration.power.startMode := 1;
   cmJRPusherAxisZ.commandConfiguration.power.stopMode := 0;
   cmJRPusherAxisZ.commandConfiguration.power.syncMotionSimulation := FALSE;
   cmJRPusherAxisZ.commandConfiguration.power.syncMotionSimulationExtendedMode := -1;
   cmJRPusherAxisZ.commandConfiguration.jog.velocity := 0.0;
   cmJRPusherAxisZ.commandConfiguration.jog.acceleration := -1.0;
   cmJRPusherAxisZ.commandConfiguration.jog.deceleration := -1.0;
   cmJRPusherAxisZ.commandConfiguration.jog.jerk := -1.0;
   cmJRPusherAxisZ.commandConfiguration.jog.positionControlled := TRUE;
   cmJRPusherAxisZ.commandConfiguration.jog.increment := 0.0;
   cmJRPusherAxisZ.commandConfiguration.jog.mode := 0;
   cmJRPusherAxisZ.commandConfiguration.moveVelocity.velocity := 0.0;
   cmJRPusherAxisZ.commandConfiguration.moveVelocity.acceleration := -1.0;
   cmJRPusherAxisZ.commandConfiguration.moveVelocity.deceleration := -1.0;
   cmJRPusherAxisZ.commandConfiguration.moveVelocity.jerk := -1.0;
   cmJRPusherAxisZ.commandConfiguration.moveVelocity.direction := 0;
   cmJRPusherAxisZ.commandConfiguration.moveVelocity.positionControlled := TRUE;
   cmJRPusherAxisZ.commandConfiguration.moveVelocity.velocityChangeOnTheFly := FALSE;
   cmJRPusherAxisZ.commandConfiguration.stop.deceleration := -1.0;
   cmJRPusherAxisZ.commandConfiguration.stop.jerk := -1.0;
   cmJRPusherAxisZ.commandConfiguration.stop.abortAcceleration := FALSE;
   cmJRPusherAxisZ.commandConfiguration.fastStop.deceleration := -1.0;
   cmJRPusherAxisZ.commandConfiguration.fastStop.jerk := -1.0;
   cmJRPusherAxisZ.commandConfiguration.fastStop.abortAcceleration := FALSE;
   cmJRPusherAxisZ.commandConfiguration.fastStop.replaceStopPossible := FALSE;
   cmJRPusherAxisZ.commandConfiguration.torqueLimiting.limit := -1.0;
   cmJRPusherAxisZ.commandConfiguration.torqueLimiting.mode := 0;
   cmJRPusherAxisZ.commandConfiguration.homing.position := 0.0;
   cmJRPusherAxisZ.commandConfiguration.homing.mode := 0;
   cmJRPusherAxisZ.commandConfiguration.homing.sensor := 0;
   cmJRPusherAxisZ.commandConfiguration.homing.extendedMode := -1;
   cmJRPusherAxisZ.commandConfiguration.homing.extendedModeTorqueLimit := 0.0;
   cmJRPusherAxisZ.commandConfiguration.homing.extendedModeTargetPosition := 0.0;
   cmJRPusherAxisZ.commandConfiguration.posRelative.distance := 0.0;
   cmJRPusherAxisZ.commandConfiguration.posRelative.velocity := -1.0;
   cmJRPusherAxisZ.commandConfiguration.posRelative.acceleration := -1.0;
   cmJRPusherAxisZ.commandConfiguration.posRelative.deceleration := -1.0;
   cmJRPusherAxisZ.commandConfiguration.posRelative.jerk := -1.0;
   cmJRPusherAxisZ.commandConfiguration.posRelative.direction := 0;
   cmJRPusherAxisZ.commandConfiguration.posAbsolute.position := 0.0;
   cmJRPusherAxisZ.commandConfiguration.posAbsolute.velocity := -1.0;
   cmJRPusherAxisZ.commandConfiguration.posAbsolute.acceleration := -1.0;
   cmJRPusherAxisZ.commandConfiguration.posAbsolute.deceleration := -1.0;
   cmJRPusherAxisZ.commandConfiguration.posAbsolute.jerk := -1.0;
   cmJRPusherAxisZ.commandConfiguration.posAbsolute.direction := 1;
   cmJRPusherAxisZ.commandConfiguration.posAbsolute.positionChangeOnTheFly := FALSE;
   cmJRPusherAxisZ.commandConfiguration.posAbsolute.velocityChangeOnTheFly := FALSE;
   cmJRPusherAxisZ.commandConfiguration.posSuperimposed.distance := 0.0;
   cmJRPusherAxisZ.commandConfiguration.posSuperimposed.velocityDiff := -1.0;
   cmJRPusherAxisZ.commandConfiguration.posSuperimposed.acceleration := -1.0;
   cmJRPusherAxisZ.commandConfiguration.posSuperimposed.deceleration := -1.0;
   cmJRPusherAxisZ.commandConfiguration.posSuperimposed.jerk := -1.0;
   cmJRPusherAxisZ.commandConfiguration.posSuperimposed.direction := 0;
   cmJRPusherAxisZ.commandConfiguration.haltSuperimposed.deceleration := -1.0;
   cmJRPusherAxisZ.commandConfiguration.haltSuperimposed.jerk := -1.0;
   cmJRPusherAxisZ.commandConfiguration.haltSuperimposed.abortAcceleration := FALSE;
   cmJRPusherAxisZ.commandConfiguration.gearInRelative.ratioNumerator := 1;
   cmJRPusherAxisZ.commandConfiguration.gearInRelative.ratioDenominator := 1;
   cmJRPusherAxisZ.commandConfiguration.gearInRelative.acceleration := -1.0;
   cmJRPusherAxisZ.commandConfiguration.gearInRelative.deceleration := -1.0;
   cmJRPusherAxisZ.commandConfiguration.gearInRelative.jerk := -1.0;
   cmJRPusherAxisZ.commandConfiguration.gearInRelative.ratioChangeOnTheFly := FALSE;
   cmJRPusherAxisZ.commandConfiguration.gearInAbsolute.ratioNumerator := 1;
   cmJRPusherAxisZ.commandConfiguration.gearInAbsolute.ratioDenominator := 1;
   cmJRPusherAxisZ.commandConfiguration.gearInAbsolute.masterSyncPosition := 0.0;
   cmJRPusherAxisZ.commandConfiguration.gearInAbsolute.slaveSyncPosition := 0.0;
   cmJRPusherAxisZ.commandConfiguration.gearInAbsolute.syncProfileReference := 1;
   cmJRPusherAxisZ.commandConfiguration.gearInAbsolute.masterStartDistance := 0.0;
   cmJRPusherAxisZ.commandConfiguration.gearInAbsolute.velocity := -1.0;
   cmJRPusherAxisZ.commandConfiguration.gearInAbsolute.acceleration := -1.0;
   cmJRPusherAxisZ.commandConfiguration.gearInAbsolute.deceleration := -1.0;
   cmJRPusherAxisZ.commandConfiguration.gearInAbsolute.jerk := -1.0;
   cmJRPusherAxisZ.commandConfiguration.gearInAbsolute.syncDirection := 1;
   cmJRPusherAxisZ.commandConfiguration.gearInAbsolute.ratioChangeOnTheFly := FALSE;
   cmJRPusherAxisZ.commandConfiguration.gearInVelocity.continuousUpdate := FALSE;
   cmJRPusherAxisZ.commandConfiguration.gearInVelocity.ratioNumerator := 1;
   cmJRPusherAxisZ.commandConfiguration.gearInVelocity.ratioDenominator := 1;
   cmJRPusherAxisZ.commandConfiguration.gearInVelocity.acceleration := -1.0;
   cmJRPusherAxisZ.commandConfiguration.gearInVelocity.deceleration := -1.0;
   cmJRPusherAxisZ.commandConfiguration.gearInVelocity.jerk := -1.0;
   cmJRPusherAxisZ.commandConfiguration.gearInVelocity.positionControlled := FALSE;
   cmJRPusherAxisZ.commandConfiguration.camIn.masterOffset := 0.0;
   cmJRPusherAxisZ.commandConfiguration.camIn.slaveOffset := 0.0;
   cmJRPusherAxisZ.commandConfiguration.camIn.masterScaling := 1.0;
   cmJRPusherAxisZ.commandConfiguration.camIn.slaveScaling := 1.0;
   cmJRPusherAxisZ.commandConfiguration.camIn.masterSyncPosition := 0.0;
   cmJRPusherAxisZ.commandConfiguration.camIn.syncProfileReference := 1;
   cmJRPusherAxisZ.commandConfiguration.camIn.masterStartDistance := 0.0;
   cmJRPusherAxisZ.commandConfiguration.camIn.velocity := -1.0;
   cmJRPusherAxisZ.commandConfiguration.camIn.acceleration := -1.0;
   cmJRPusherAxisZ.commandConfiguration.camIn.deceleration := -1.0;
   cmJRPusherAxisZ.commandConfiguration.camIn.jerk := -1.0;
   cmJRPusherAxisZ.commandConfiguration.camIn.applicationMode := 0;
   cmJRPusherAxisZ.commandConfiguration.camIn.syncDirection := 1;
   cmJRPusherAxisZ.commandConfiguration.gearOutCamOut.slavePosition := 0.0;
   cmJRPusherAxisZ.commandConfiguration.gearOutCamOut.syncProfileReference := 1;
   cmJRPusherAxisZ.commandConfiguration.gearOutCamOut.masterStopDistance := 0.0;
   cmJRPusherAxisZ.commandConfiguration.gearOutCamOut.deceleration := -1.0;
   cmJRPusherAxisZ.commandConfiguration.gearOutCamOut.jerk := -1.0;
   cmJRPusherAxisZ.commandConfiguration.gearOutCamOut.syncOutDirection := 3;
   cmJRPusherAxisZ.commandConfiguration.gearOutCamOut.gearOutCamOutMode := -1;
   cmJRPusherAxisZ.commandConfiguration.phasing.phaseShift := 0.0;
   cmJRPusherAxisZ.commandConfiguration.phasing.velocity := -1.0;
   cmJRPusherAxisZ.commandConfiguration.phasing.acceleration := -1.0;
   cmJRPusherAxisZ.commandConfiguration.phasing.deceleration := -1.0;
   cmJRPusherAxisZ.commandConfiguration.phasing.jerk := -1.0;
   cmJRPusherAxisZ.commandConfiguration.phasing.profileReference := 0;
   cmJRPusherAxisZ.commandConfiguration.phasing.phasingDistance := 0.0;
   cmJRPusherAxisZ.commandConfiguration.phasing.startPosition := 0.0;
   cmJRPusherAxisZ.commandConfiguration.phasing.direction := 3;
   cmJRPusherAxisZ.commandConfiguration.phasing.phaseAbsolute := TRUE;
   cmJRPusherAxisZ.commandConfiguration.phasing.phaseShiftChangeOnTheFly := FALSE;
   cmJRPusherAxisZ.commandConfiguration.offset.offset := 0.0;
   cmJRPusherAxisZ.commandConfiguration.offset.profileReference := 1;
   cmJRPusherAxisZ.commandConfiguration.offset.offsetDistance := 0.0;
   cmJRPusherAxisZ.commandConfiguration.offset.startPosition := 0.0;
   cmJRPusherAxisZ.commandConfiguration.offset.direction := 3;
   cmJRPusherAxisZ.commandConfiguration.offset.offsetAbsolute := TRUE;
   cmJRPusherAxisZ.commandConfiguration.offset.offsetChangeOnTheFly := FALSE;
   cmJRPusherAxisZ.commands.enableMasterControl := TRUE;
   cmJRPusherAxisZ.commands.enableAxis := FALSE;
   cmJRPusherAxisZ.commands.resetAxis := FALSE;
   cmJRPusherAxisZ.commands.openBrake := FALSE;
   cmJRPusherAxisZ.commands.jogForward := FALSE;
   cmJRPusherAxisZ.commands.jogBackward := FALSE;
   cmJRPusherAxisZ.commands.moveVelocity := FALSE;
   cmJRPusherAxisZ.commands.stop := FALSE;
   cmJRPusherAxisZ.commands.fastStop := FALSE;
   cmJRPusherAxisZ.commands.torqueLimiting := FALSE;
   cmJRPusherAxisZ.commands.homing := FALSE;
   cmJRPusherAxisZ.commands.posRelative := FALSE;
   cmJRPusherAxisZ.commands.posAbsolute := FALSE;
   cmJRPusherAxisZ.commands.posSuperimposed := FALSE;
   cmJRPusherAxisZ.commands.haltSuperimposed := FALSE;
   cmJRPusherAxisZ.commands.selectSetPosition := -1;
   cmJRPusherAxisZ.commands.uploadParameters := FALSE;
   cmJRPusherAxisZ.commands.refreshConfiguration := FALSE;
   cmJRPusherAxisZ.commands.editConfiguration := FALSE;
   cmJRPusherAxisZ.commands.saveConfiguration := FALSE;
   cmJRPusherAxisZ.commands.uploadCurrentTorque := FALSE;
   cmJRPusherAxisZ.commands.reset := FALSE;
   cmJRPusherAxisZ.monitoring.enable := TRUE;
   cmJRPusherAxisZ.monitoring.referenceDesignator := WSTRING#'JRPusherAxisZ';
   cmJRPusherAxisZ.monitoring.enabled := TRUE;
   cmJRPusherAxisZ.monitoring.enableManualCmds := FALSE;
   cmJRPusherAxisZ.monitoring.reset := FALSE;
   cmJRPusherAxisZ.monitoring.resetAxis := FALSE;
   cmJRPusherAxisZ.monitoring.enableAxis := TRUE;
   cmJRPusherAxisZ.monitoring.openBrake := FALSE;
   cmJRPusherAxisZ.monitoring.jogBackward := FALSE;
   cmJRPusherAxisZ.monitoring.jogForward := FALSE;
   cmJRPusherAxisZ.monitoring.moveVelocity := FALSE;
   cmJRPusherAxisZ.monitoring.stop := FALSE;
   cmJRPusherAxisZ.monitoring.fastStop := FALSE;
   cmJRPusherAxisZ.monitoring.torqueLimiting := FALSE;
   cmJRPusherAxisZ.monitoring.homing := FALSE;
   cmJRPusherAxisZ.monitoring.posRelative := FALSE;
   cmJRPusherAxisZ.monitoring.posAbsolute := FALSE;
   cmJRPusherAxisZ.monitoring.posSuperimposed := FALSE;
   cmJRPusherAxisZ.monitoring.haltSuperimposed := FALSE;
   cmJRPusherAxisZ.monitoring.brakeOpened := FALSE;
   cmJRPusherAxisZ.monitoring.axisEnabled := TRUE;
   cmJRPusherAxisZ.monitoring.resetActive := FALSE;
   cmJRPusherAxisZ.monitoring.inVelocity := FALSE;
   cmJRPusherAxisZ.monitoring.inLimitation := FALSE;
   cmJRPusherAxisZ.monitoring.inClamping := FALSE;
   cmJRPusherAxisZ.monitoring.startSync := FALSE;
   cmJRPusherAxisZ.monitoring.inSync := FALSE;
   cmJRPusherAxisZ.monitoring.inSimulation := FALSE;
   cmJRPusherAxisZ.monitoring.jogSelected := FALSE;
   cmJRPusherAxisZ.monitoring.moveVelocitySelected := FALSE;
   cmJRPusherAxisZ.monitoring.stopSelected := FALSE;
   cmJRPusherAxisZ.monitoring.fastStopSelected := FALSE;
   cmJRPusherAxisZ.monitoring.torqueLimitingSelected := FALSE;
   cmJRPusherAxisZ.monitoring.homingSelected := FALSE;
   cmJRPusherAxisZ.monitoring.posRelativeSelected := FALSE;
   cmJRPusherAxisZ.monitoring.posAbsoluteSelected := FALSE;
   cmJRPusherAxisZ.monitoring.posSuperimposedSelected := FALSE;
   cmJRPusherAxisZ.monitoring.haltSuperimposedSelected := FALSE;
   cmJRPusherAxisZ.monitoring.commandBusy := FALSE;
   cmJRPusherAxisZ.monitoring.commandDone := FALSE;
   cmJRPusherAxisZ.monitoring.commandAborted := FALSE;
   cmJRPusherAxisZ.monitoring.homingCommandBusy := FALSE;
   cmJRPusherAxisZ.monitoring.homingCommandDone := FALSE;
   cmJRPusherAxisZ.monitoring.homingCommandAborted := FALSE;
   cmJRPusherAxisZ.monitoring.superimposedBusy := FALSE;
   cmJRPusherAxisZ.monitoring.superimposedDone := FALSE;
   cmJRPusherAxisZ.monitoring.superimposedAborted := FALSE;
   cmJRPusherAxisZ.monitoring.selectSetPosition := -1;
   cmJRPusherAxisZ.monitoring.selectionController := FALSE;
   cmJRPusherAxisZ.monitoring.interlockGeneral := TRUE;
   cmJRPusherAxisZ.monitoring.interlockJogForward := TRUE;
   cmJRPusherAxisZ.monitoring.interlockJogBackward := TRUE;
   cmJRPusherAxisZ.monitoring.interlockWarningGeneral := FALSE;
   cmJRPusherAxisZ.monitoring.interlockWarningJogForward := FALSE;
   cmJRPusherAxisZ.monitoring.interlockWarningJogBackward := FALSE;
   cmJRPusherAxisZ.monitoring.valid := TRUE;
   cmJRPusherAxisZ.monitoring.busy := TRUE;
   cmJRPusherAxisZ.monitoring.error := FALSE;
   cmJRPusherAxisZ.monitoring.status := 16#7002;
   cmJRPusherAxisZ.monitoring.subfunctionStatus := 16#0000;
   cmJRPusherAxisZ.monitoring.actualPosition := 0.0;
   cmJRPusherAxisZ.monitoring.actualSpeed := 0.0;
   cmJRPusherAxisZ.monitoring.speedUnit := 1062;
   cmJRPusherAxisZ.monitoring.positionUnit := 1013;
   cmJRPusherAxisZ.monitoring.axisStatus1 := 16#0200_10E1;
   cmJRPusherAxisZ.monitoring.axisStatus2 := 16#0000_0000;
   cmJRPusherAxisZ.monitoring.axisType := 1;
   cmJRPusherAxisZ.monitoring.maxVelocity := 500.0;
   cmJRPusherAxisZ.monitoring.actualCurrent := 0.0;
   cmJRPusherAxisZ.monitoring.actualTorque := 0.0;
   cmJRPusherAxisZ.monitoring.velocityOverrideEnabled := FALSE;
   cmJRPusherAxisZ.monitoring.sinaParaError := FALSE;
   cmJRPusherAxisZ.monitoring.sinaParaStatus := 16#0000_0000;
   cmJRPusherAxisZ.configuration.referenceDesignator := WSTRING#'JRPusherAxisZ';
   cmJRPusherAxisZ.configuration.disableAlarms := FALSE;
   cmJRPusherAxisZ.configuration.masterControlPopUp := TRUE;
   cmJRPusherAxisZ.configuration.setPositions[0].position := 0.0;
   cmJRPusherAxisZ.configuration.setPositions[1].position := 100.0;
   cmJRPusherAxisZ.configuration.setPositions[2].position := 0.0;
   cmJRPusherAxisZ.configuration.setPositions[3].position := 100.0;
   cmJRPusherAxisZ.configuration.setPositions[4..15].position := 0.0;
   cmJRPusherAxisZ.configuration.setPositions[0..3].velocity := 100.0;
   cmJRPusherAxisZ.configuration.setPositions[4..15].velocity := -1.0;
   cmJRPusherAxisZ.configuration.setPositions[0..3].acceleration := 1000.0;
   cmJRPusherAxisZ.configuration.setPositions[4..15].acceleration := -1.0;
   cmJRPusherAxisZ.configuration.setPositions[0..3].deceleration := 1000.0;
   cmJRPusherAxisZ.configuration.setPositions[4..15].deceleration := -1.0;
   cmJRPusherAxisZ.configuration.setPositions[0..15]."name" := '';
   cmSepaCutterUpDown.commands.refreshConfiguration := FALSE;
   cmSepaCutterUpDown.commands.editConfiguration := FALSE;
   cmSepaCutterUpDown.commands.saveConfiguration := FALSE;
   cmSepaCutterUpDown.commands.reset := FALSE;
   cmSepaCutterUpDown.commands.commandHomePos := FALSE;
   cmSepaCutterUpDown.commands.commandWorkPos := FALSE;
   cmSepaCutterUpDown.monitoring.enable := TRUE;
   cmSepaCutterUpDown.monitoring.referenceDesignator := WSTRING#'SepaCutterUpDown';
   cmSepaCutterUpDown.monitoring.commandHomePos := FALSE;
   cmSepaCutterUpDown.monitoring.commandWorkPos := FALSE;
   cmSepaCutterUpDown.monitoring.goToHomePos := TRUE;
   cmSepaCutterUpDown.monitoring.goToWorkPos := FALSE;
   cmSepaCutterUpDown.monitoring.inHomePos := TRUE;
   cmSepaCutterUpDown.monitoring.inWorkPos := FALSE;
   cmSepaCutterUpDown.monitoring.reset := FALSE;
   cmSepaCutterUpDown.monitoring.enableManualCmds := FALSE;
   cmSepaCutterUpDown.monitoring.error := FALSE;
   cmSepaCutterUpDown.monitoring.interlockHomePos := TRUE;
   cmSepaCutterUpDown.monitoring.interlockWorkPos := TRUE;
   cmSepaCutterUpDown.monitoring.status := 16#7004;
   cmSepaCutterUpDown.monitoring.interlockWarningWorkPos := FALSE;
   cmSepaCutterUpDown.monitoring.interlockWarningHomePos := FALSE;
   cmSepaCutterUpDown.configuration.referenceDesignator := WSTRING#'SepaCutterUpDown';
   cmSepaCutterUpDown.configuration.monitoringLeavingFeedback := T#5S;
   cmSepaCutterUpDown.configuration.monitoringReachingFeedback := T#5S;
   cmSepaCutterUpDown.configuration.monitoringDiscrepancy := T#0MS;
   cmSepaCutterUpDown.configuration.setOutputHomeContinuously := TRUE;
   cmSepaCutterUpDown.configuration.setOutputWorkContinuously := TRUE;
   cmSepaCutterUpDown.configuration.disableHomeCommand := FALSE;
   cmSepaCutterUpDown.configuration.disableFeedbackHomePos := FALSE;
   cmSepaCutterUpDown.configuration.disableFeedbackWorkPos := FALSE;
   cmSepaCutterUpDown.configuration.disableAlarms := FALSE;
   cmSepaCutterUpDown.configuration.resetOutputsOnError := FALSE;
   cmSepaCutterUpDown.configuration.allwaysWaitOnReachingTime := FALSE;
   cmSepaClampTopUpDown.commands.refreshConfiguration := FALSE;
   cmSepaClampTopUpDown.commands.editConfiguration := FALSE;
   cmSepaClampTopUpDown.commands.saveConfiguration := FALSE;
   cmSepaClampTopUpDown.commands.reset := FALSE;
   cmSepaClampTopUpDown.commands.commandHomePos := FALSE;
   cmSepaClampTopUpDown.commands.commandWorkPos := FALSE;
   cmSepaClampTopUpDown.monitoring.enable := TRUE;
   cmSepaClampTopUpDown.monitoring.referenceDesignator := WSTRING#'SepaClampTopUpDown';
   cmSepaClampTopUpDown.monitoring.commandHomePos := FALSE;
   cmSepaClampTopUpDown.monitoring.commandWorkPos := FALSE;
   cmSepaClampTopUpDown.monitoring.goToHomePos := FALSE;
   cmSepaClampTopUpDown.monitoring.goToWorkPos := TRUE;
   cmSepaClampTopUpDown.monitoring.inHomePos := FALSE;
   cmSepaClampTopUpDown.monitoring.inWorkPos := TRUE;
   cmSepaClampTopUpDown.monitoring.reset := FALSE;
   cmSepaClampTopUpDown.monitoring.enableManualCmds := FALSE;
   cmSepaClampTopUpDown.monitoring.error := FALSE;
   cmSepaClampTopUpDown.monitoring.interlockHomePos := TRUE;
   cmSepaClampTopUpDown.monitoring.interlockWorkPos := TRUE;
   cmSepaClampTopUpDown.monitoring.status := 16#7006;
   cmSepaClampTopUpDown.monitoring.interlockWarningWorkPos := FALSE;
   cmSepaClampTopUpDown.monitoring.interlockWarningHomePos := FALSE;
   cmSepaClampTopUpDown.configuration.referenceDesignator := WSTRING#'SepaClampTopUpDown';
   cmSepaClampTopUpDown.configuration.monitoringLeavingFeedback := T#5S;
   cmSepaClampTopUpDown.configuration.monitoringReachingFeedback := T#5S;
   cmSepaClampTopUpDown.configuration.monitoringDiscrepancy := T#0MS;
   cmSepaClampTopUpDown.configuration.setOutputHomeContinuously := TRUE;
   cmSepaClampTopUpDown.configuration.setOutputWorkContinuously := TRUE;
   cmSepaClampTopUpDown.configuration.disableHomeCommand := FALSE;
   cmSepaClampTopUpDown.configuration.disableFeedbackHomePos := FALSE;
   cmSepaClampTopUpDown.configuration.disableFeedbackWorkPos := FALSE;
   cmSepaClampTopUpDown.configuration.disableAlarms := FALSE;
   cmSepaClampTopUpDown.configuration.resetOutputsOnError := FALSE;
   cmSepaClampTopUpDown.configuration.allwaysWaitOnReachingTime := FALSE;
   cmSepaClampBottomUpDown.commands.refreshConfiguration := FALSE;
   cmSepaClampBottomUpDown.commands.editConfiguration := FALSE;
   cmSepaClampBottomUpDown.commands.saveConfiguration := FALSE;
   cmSepaClampBottomUpDown.commands.reset := FALSE;
   cmSepaClampBottomUpDown.commands.commandHomePos := FALSE;
   cmSepaClampBottomUpDown.commands.commandWorkPos := FALSE;
   cmSepaClampBottomUpDown.monitoring.enable := TRUE;
   cmSepaClampBottomUpDown.monitoring.referenceDesignator := WSTRING#'ClampBottomUpDown';
   cmSepaClampBottomUpDown.monitoring.commandHomePos := FALSE;
   cmSepaClampBottomUpDown.monitoring.commandWorkPos := FALSE;
   cmSepaClampBottomUpDown.monitoring.goToHomePos := FALSE;
   cmSepaClampBottomUpDown.monitoring.goToWorkPos := TRUE;
   cmSepaClampBottomUpDown.monitoring.inHomePos := FALSE;
   cmSepaClampBottomUpDown.monitoring.inWorkPos := TRUE;
   cmSepaClampBottomUpDown.monitoring.reset := FALSE;
   cmSepaClampBottomUpDown.monitoring.enableManualCmds := FALSE;
   cmSepaClampBottomUpDown.monitoring.error := FALSE;
   cmSepaClampBottomUpDown.monitoring.interlockHomePos := TRUE;
   cmSepaClampBottomUpDown.monitoring.interlockWorkPos := TRUE;
   cmSepaClampBottomUpDown.monitoring.status := 16#7006;
   cmSepaClampBottomUpDown.monitoring.interlockWarningWorkPos := FALSE;
   cmSepaClampBottomUpDown.monitoring.interlockWarningHomePos := FALSE;
   cmSepaClampBottomUpDown.configuration.referenceDesignator := WSTRING#'ClampBottomUpDown';
   cmSepaClampBottomUpDown.configuration.monitoringLeavingFeedback := T#5S;
   cmSepaClampBottomUpDown.configuration.monitoringReachingFeedback := T#5S;
   cmSepaClampBottomUpDown.configuration.monitoringDiscrepancy := T#0MS;
   cmSepaClampBottomUpDown.configuration.setOutputHomeContinuously := TRUE;
   cmSepaClampBottomUpDown.configuration.setOutputWorkContinuously := TRUE;
   cmSepaClampBottomUpDown.configuration.disableHomeCommand := FALSE;
   cmSepaClampBottomUpDown.configuration.disableFeedbackHomePos := FALSE;
   cmSepaClampBottomUpDown.configuration.disableFeedbackWorkPos := FALSE;
   cmSepaClampBottomUpDown.configuration.disableAlarms := FALSE;
   cmSepaClampBottomUpDown.configuration.resetOutputsOnError := FALSE;
   cmSepaClampBottomUpDown.configuration.allwaysWaitOnReachingTime := FALSE;
   cmStackGripperOpenClose.commands.refreshConfiguration := FALSE;
   cmStackGripperOpenClose.commands.editConfiguration := FALSE;
   cmStackGripperOpenClose.commands.saveConfiguration := FALSE;
   cmStackGripperOpenClose.commands.reset := FALSE;
   cmStackGripperOpenClose.commands.commandHomePos := FALSE;
   cmStackGripperOpenClose.commands.commandWorkPos := FALSE;
   cmStackGripperOpenClose.monitoring.enable := TRUE;
   cmStackGripperOpenClose.monitoring.referenceDesignator := WSTRING#'GripperOpenClose';
   cmStackGripperOpenClose.monitoring.commandHomePos := FALSE;
   cmStackGripperOpenClose.monitoring.commandWorkPos := FALSE;
   cmStackGripperOpenClose.monitoring.goToHomePos := TRUE;
   cmStackGripperOpenClose.monitoring.goToWorkPos := FALSE;
   cmStackGripperOpenClose.monitoring.inHomePos := TRUE;
   cmStackGripperOpenClose.monitoring.inWorkPos := FALSE;
   cmStackGripperOpenClose.monitoring.reset := FALSE;
   cmStackGripperOpenClose.monitoring.enableManualCmds := FALSE;
   cmStackGripperOpenClose.monitoring.error := FALSE;
   cmStackGripperOpenClose.monitoring.interlockHomePos := TRUE;
   cmStackGripperOpenClose.monitoring.interlockWorkPos := TRUE;
   cmStackGripperOpenClose.monitoring.status := 16#7004;
   cmStackGripperOpenClose.monitoring.interlockWarningWorkPos := FALSE;
   cmStackGripperOpenClose.monitoring.interlockWarningHomePos := FALSE;
   cmStackGripperOpenClose.configuration.referenceDesignator := WSTRING#'GripperOpenClose';
   cmStackGripperOpenClose.configuration.monitoringLeavingFeedback := T#5S;
   cmStackGripperOpenClose.configuration.monitoringReachingFeedback := T#5S;
   cmStackGripperOpenClose.configuration.monitoringDiscrepancy := T#0MS;
   cmStackGripperOpenClose.configuration.setOutputHomeContinuously := TRUE;
   cmStackGripperOpenClose.configuration.setOutputWorkContinuously := TRUE;
   cmStackGripperOpenClose.configuration.disableHomeCommand := FALSE;
   cmStackGripperOpenClose.configuration.disableFeedbackHomePos := FALSE;
   cmStackGripperOpenClose.configuration.disableFeedbackWorkPos := FALSE;
   cmStackGripperOpenClose.configuration.disableAlarms := FALSE;
   cmStackGripperOpenClose.configuration.resetOutputsOnError := FALSE;
   cmStackGripperOpenClose.configuration.allwaysWaitOnReachingTime := FALSE;
   cmStackGripperFwdBwd.commands.refreshConfiguration := FALSE;
   cmStackGripperFwdBwd.commands.editConfiguration := FALSE;
   cmStackGripperFwdBwd.commands.saveConfiguration := FALSE;
   cmStackGripperFwdBwd.commands.reset := FALSE;
   cmStackGripperFwdBwd.commands.commandHomePos := FALSE;
   cmStackGripperFwdBwd.commands.commandWorkPos := FALSE;
   cmStackGripperFwdBwd.monitoring.enable := TRUE;
   cmStackGripperFwdBwd.monitoring.referenceDesignator := WSTRING#'GripperFwdBwd';
   cmStackGripperFwdBwd.monitoring.commandHomePos := FALSE;
   cmStackGripperFwdBwd.monitoring.commandWorkPos := FALSE;
   cmStackGripperFwdBwd.monitoring.goToHomePos := TRUE;
   cmStackGripperFwdBwd.monitoring.goToWorkPos := FALSE;
   cmStackGripperFwdBwd.monitoring.inHomePos := TRUE;
   cmStackGripperFwdBwd.monitoring.inWorkPos := FALSE;
   cmStackGripperFwdBwd.monitoring.reset := FALSE;
   cmStackGripperFwdBwd.monitoring.enableManualCmds := FALSE;
   cmStackGripperFwdBwd.monitoring.error := FALSE;
   cmStackGripperFwdBwd.monitoring.interlockHomePos := TRUE;
   cmStackGripperFwdBwd.monitoring.interlockWorkPos := TRUE;
   cmStackGripperFwdBwd.monitoring.status := 16#7004;
   cmStackGripperFwdBwd.monitoring.interlockWarningWorkPos := FALSE;
   cmStackGripperFwdBwd.monitoring.interlockWarningHomePos := FALSE;
   cmStackGripperFwdBwd.configuration.referenceDesignator := WSTRING#'GripperFwdBwd';
   cmStackGripperFwdBwd.configuration.monitoringLeavingFeedback := T#5S;
   cmStackGripperFwdBwd.configuration.monitoringReachingFeedback := T#5S;
   cmStackGripperFwdBwd.configuration.monitoringDiscrepancy := T#0MS;
   cmStackGripperFwdBwd.configuration.setOutputHomeContinuously := TRUE;
   cmStackGripperFwdBwd.configuration.setOutputWorkContinuously := TRUE;
   cmStackGripperFwdBwd.configuration.disableHomeCommand := FALSE;
   cmStackGripperFwdBwd.configuration.disableFeedbackHomePos := FALSE;
   cmStackGripperFwdBwd.configuration.disableFeedbackWorkPos := FALSE;
   cmStackGripperFwdBwd.configuration.disableAlarms := FALSE;
